C05467=1046.708,-58.246,426.994,169.791,33.093,156.253
C05468=1046.701,-58.495,427.006,169.789,33.092,156.253
C05469=1046.696,-58.746,427.017,169.787,33.091,156.252
C05470=1046.689,-58.995,427.029,169.784,33.090,156.252
C05471=1046.683,-59.245,427.041,169.782,33.089,156.252
C05472=1046.677,-59.495,427.054,169.780,33.088,156.252
C05473=1046.671,-59.744,427.065,169.778,33.088,156.252
C05474=1046.664,-59.993,427.077,169.776,33.086,156.252
C05475=1046.658,-60.243,427.090,169.774,33.085,156.252
C05476=1046.651,-60.493,427.102,169.772,33.085,156.252
C05477=1046.645,-60.742,427.114,169.769,33.084,156.252
C05478=1046.639,-60.992,427.126,169.767,33.082,156.252
C05479=1046.633,-61.242,427.137,169.765,33.081,156.252
C05480=1046.626,-61.491,427.149,169.763,33.081,156.251
C05481=1046.621,-61.741,427.162,169.761,33.080,156.251
C05482=1046.614,-61.991,427.174,169.759,33.079,156.251
C05483=1046.607,-62.240,427.186,169.757,33.078,156.251
C05484=1046.602,-62.489,427.198,169.755,33.077,156.251
C05485=1046.596,-62.740,427.209,169.752,33.076,156.251
C05486=1046.589,-62.989,427.221,169.750,33.075,156.251
C05487=1046.583,-63.239,427.234,169.748,33.074,156.251
C05488=1046.576,-63.489,427.246,169.746,33.073,156.251
C05489=1046.570,-63.737,427.257,169.744,33.072,156.251
C05490=1046.565,-63.988,427.269,169.742,33.071,156.251
C05491=1046.558,-64.238,427.281,169.739,33.070,156.250
C05492=1046.551,-64.487,427.293,169.738,33.069,156.250
C05493=1046.545,-64.736,427.305,169.736,33.068,156.250
C05494=1046.540,-64.986,427.316,169.734,33.067,156.250
C05495=1046.533,-65.236,427.328,169.732,33.066,156.250
C05496=1046.527,-65.485,427.340,169.730,33.065,156.250
C05497=1046.521,-65.735,427.353,169.728,33.065,156.250
C05498=1046.515,-65.985,427.364,169.725,33.064,156.250
C05499=1046.508,-66.235,427.376,169.723,33.062,156.250
C05500=1046.503,-66.484,427.388,169.721,33.061,156.250
C05501=1046.497,-66.734,427.399,169.719,33.061,156.250
C05502=1046.489,-67.016,427.413,169.716,33.060,156.250
C05503=1046.483,-67.299,427.426,169.714,33.058,156.249
C05504=1046.476,-67.581,427.440,169.712,33.057,156.249
C05505=1046.469,-67.863,427.453,169.709,33.057,156.249
C05506=1046.462,-68.113,427.465,169.707,33.056,156.249
C05507=1046.456,-68.362,427.476,169.705,33.055,156.249
C05508=1046.450,-68.612,427.487,169.703,33.054,156.249
C05509=1046.444,-68.862,427.500,169.701,33.053,156.249
C05510=1046.438,-69.111,427.511,169.698,33.052,156.249
C05511=1046.432,-69.361,427.523,169.696,33.051,156.249
C05512=1046.425,-69.611,427.535,169.694,33.050,156.249
C05513=1046.420,-69.860,427.546,169.692,33.049,156.249
C05514=1046.413,-70.110,427.558,169.690,33.049,156.248
C05515=1046.407,-70.360,427.569,169.688,33.048,156.248
C05516=1046.401,-70.609,427.581,169.685,33.047,156.248
C05517=1046.395,-70.859,427.593,169.683,33.046,156.248
C05518=1046.389,-71.108,427.604,169.681,33.045,156.248
C05519=1046.383,-71.358,427.616,169.679,33.044,156.248
C05520=1046.376,-71.608,427.628,169.677,33.043,156.248
C05521=1046.371,-71.857,427.640,169.674,33.042,156.248
C05522=1046.365,-72.107,427.651,169.672,33.041,156.248
C05523=1046.359,-72.356,427.663,169.670,33.040,156.248
C05524=1046.352,-72.607,427.674,169.669,33.040,156.248
C05525=1046.347,-72.856,427.686,169.667,33.039,156.248
C05526=1046.341,-73.106,427.697,169.665,33.038,156.248
C05527=1046.334,-73.356,427.709,169.662,33.037,156.248
C05528=1046.328,-73.605,427.720,169.660,33.036,156.247
C05529=1046.322,-73.855,427.731,169.658,33.035,156.247
C05530=1046.317,-74.104,427.744,169.656,33.035,156.247
C05531=1046.310,-74.355,427.755,169.654,33.034,156.247
C05532=1046.304,-74.603,427.766,169.651,33.033,156.247
C05533=1046.298,-74.854,427.778,169.649,33.032,156.247
C05534=1046.292,-75.104,427.789,169.647,33.031,156.247
C05535=1046.285,-75.352,427.800,169.645,33.030,156.247
C05536=1046.278,-75.603,427.811,169.643,33.030,156.247
C05537=1046.273,-75.852,427.822,169.640,33.029,156.247
C05538=1046.266,-76.102,427.834,169.638,33.028,156.247
C05539=1046.260,-76.351,427.845,169.636,33.028,156.247
C05540=1046.254,-76.601,427.856,169.634,33.027,156.247
C05541=1046.248,-76.850,427.868,169.632,33.026,156.247
C05542=1046.242,-77.100,427.879,169.629,33.025,156.247
C05543=1046.235,-77.351,427.890,169.627,33.024,156.247
C05544=1046.229,-77.599,427.902,169.625,33.024,156.247
C05545=1046.223,-77.850,427.913,169.623,33.023,156.247
C05546=1046.217,-78.099,427.924,169.620,33.022,156.247
C05547=1046.210,-78.349,427.936,169.618,33.021,156.246
C05548=1046.205,-78.598,427.947,169.616,33.021,156.246
C05549=1046.198,-78.848,427.958,169.614,33.020,156.246
C05550=1046.193,-79.098,427.969,169.612,33.020,156.246
C05551=1046.186,-79.348,427.980,169.609,33.019,156.246
C05552=1046.180,-79.597,427.992,169.607,33.018,156.246
C05553=1046.174,-79.847,428.003,169.605,33.017,156.246
C05554=1046.167,-80.096,428.013,169.603,33.016,156.246
C05555=1046.161,-80.346,428.025,169.601,33.016,156.246
C05556=1046.155,-80.596,428.035,169.599,33.015,156.246
C05557=1046.149,-80.846,428.047,169.597,33.014,156.246
C05558=1046.142,-81.095,428.058,169.595,33.014,156.246
C05559=1046.136,-81.345,428.069,169.592,33.013,156.246
C05560=1046.130,-81.594,428.080,169.590,33.012,156.246
C05561=1046.124,-81.845,428.091,169.588,33.012,156.246
C05562=1046.117,-82.094,428.101,169.586,33.011,156.246
C05563=1046.111,-82.344,428.113,169.583,33.011,156.246
C05564=1046.105,-82.593,428.123,169.581,33.010,156.246
C05565=1046.098,-82.843,428.134,169.579,33.009,156.246
C05566=1046.091,-83.127,428.147,169.576,33.009,156.246
C05567=1046.084,-83.412,428.160,169.574,33.008,156.246
C05568=1046.077,-83.697,428.172,169.571,33.007,156.246
C05569=1046.070,-83.981,428.184,169.569,33.007,156.246
C05570=1046.063,-84.231,428.196,169.566,33.006,156.246
C05571=1046.058,-84.480,428.206,169.564,33.006,156.246
C05572=1046.051,-84.730,428.217,169.562,33.005,156.246
C05573=1046.045,-84.980,428.228,169.560,33.005,156.246
C05574=1046.039,-85.229,428.239,169.557,33.004,156.246
C05575=1046.032,-85.479,428.249,169.555,33.003,156.246
C05576=1046.026,-85.729,428.260,169.553,33.003,156.246
C05577=1046.020,-85.979,428.272,169.551,33.002,156.246
C05578=1046.013,-86.228,428.282,169.548,33.002,156.246
C05579=1046.008,-86.477,428.293,169.546,33.001,156.246
C05580=1046.001,-86.728,428.304,169.544,33.000,156.246
C05581=1045.995,-86.977,428.314,169.542,33.000,156.246
C05582=1045.989,-87.227,428.326,169.540,32.999,156.246
C05583=1045.983,-87.477,428.336,169.538,32.999,156.245
C05584=1045.977,-87.726,428.346,169.536,32.998,156.246
C05585=1045.970,-87.977,428.357,169.533,32.997,156.245
C05586=1045.965,-88.226,428.368,169.531,32.997,156.246
C05587=1045.958,-88.475,428.378,169.529,32.996,156.245
C05588=1045.952,-88.725,428.390,169.527,32.996,156.246
C05589=1045.946,-88.975,428.400,169.524,32.995,156.245
C05590=1045.940,-89.224,428.411,169.522,32.995,156.245
C05591=1045.933,-89.474,428.422,169.520,32.994,156.245
C05592=1045.927,-89.724,428.433,169.518,32.994,156.245
C05593=1045.921,-89.974,428.442,169.515,32.993,156.245
C05594=1045.915,-90.224,428.454,169.513,32.993,156.245
C05595=1045.909,-90.473,428.465,169.511,32.992,156.245
C05596=1045.903,-90.722,428.475,169.508,32.992,156.245
C05597=1045.896,-90.973,428.486,169.506,32.991,156.245
C05598=1045.890,-91.222,428.496,169.504,32.991,156.245
C05599=1045.884,-91.472,428.507,169.502,32.990,156.245
C05600=1045.878,-91.722,428.518,169.499,32.990,156.245
C05601=1045.872,-91.971,428.528,169.497,32.989,156.245
C05602=1045.866,-92.221,428.539,169.495,32.989,156.245
C05603=1045.860,-92.470,428.550,169.493,32.988,156.245
C05604=1045.853,-92.721,428.560,169.490,32.988,156.245
C05605=1045.848,-92.970,428.571,169.488,32.987,156.245
C05606=1045.841,-93.219,428.581,169.486,32.987,156.245
C05607=1045.835,-93.469,428.592,169.483,32.986,156.245
C05608=1045.829,-93.720,428.602,169.481,32.986,156.245
C05609=1045.823,-93.969,428.613,169.479,32.985,156.245
C05610=1045.817,-94.218,428.623,169.477,32.985,156.245
C05611=1045.811,-94.468,428.633,169.475,32.984,156.245
C05612=1045.805,-94.718,428.644,169.473,32.983,156.245
C05613=1045.799,-94.968,428.655,169.471,32.983,156.245
C05614=1045.792,-95.217,428.665,169.468,32.982,156.245
C05615=1045.787,-95.467,428.676,169.466,32.982,156.245
C05616=1045.781,-95.716,428.686,169.464,32.982,156.245
C05617=1045.775,-95.966,428.697,169.462,32.981,156.245
C05618=1045.769,-96.217,428.707,169.459,32.981,156.245
C05619=1045.762,-96.466,428.718,169.457,32.980,156.245
C05620=1045.757,-96.716,428.728,169.455,32.980,156.245
C05621=1045.750,-96.965,428.738,169.452,32.980,156.245
C05622=1045.745,-97.215,428.749,169.450,32.979,156.245
C05623=1045.738,-97.465,428.759,169.448,32.979,156.245
C05624=1045.732,-97.715,428.770,169.446,32.978,156.245
C05625=1045.726,-97.964,428.779,169.443,32.977,156.245
C05626=1045.720,-98.214,428.790,169.441,32.977,156.245
C05627=1045.714,-98.463,428.800,169.439,32.977,156.246
C05628=1045.707,-98.714,428.810,169.436,32.977,156.246
C05629=1045.701,-98.963,428.821,169.434,32.977,156.246
C05630=1045.695,-99.250,428.832,169.431,32.976,156.246
C05631=1045.687,-99.536,428.844,169.429,32.975,156.246
C05632=1045.680,-99.824,428.855,169.426,32.975,156.246
C05633=1045.673,-100.111,428.868,169.423,32.975,156.246
C05634=1045.667,-100.360,428.877,169.421,32.974,156.246
C05635=1045.660,-100.610,428.888,169.419,32.974,156.246
C05636=1045.655,-100.860,428.898,169.416,32.974,156.246
C05637=1045.648,-101.109,428.908,169.415,32.973,156.246
C05638=1045.642,-101.359,428.918,169.413,32.973,156.246
C05639=1045.636,-101.608,428.929,169.410,32.973,156.246
C05640=1045.629,-101.859,428.939,169.408,32.972,156.246
C05641=1045.623,-102.108,428.949,169.406,32.972,156.246
C05642=1045.618,-102.358,428.959,169.403,32.972,156.246
C05643=1045.611,-102.608,428.969,169.401,32.971,156.246
C05644=1045.605,-102.857,428.979,169.399,32.971,156.246
C05645=1045.600,-103.107,428.989,169.397,32.971,156.246
C05646=1045.593,-103.356,428.999,169.394,32.971,156.246
C05647=1045.587,-103.606,429.009,169.392,32.970,156.246
C05648=1045.581,-103.856,429.018,169.390,32.970,156.246
C05649=1045.575,-104.105,429.029,169.387,32.969,156.246
C05650=1045.569,-104.355,429.039,169.385,32.969,156.246
C05651=1045.562,-104.606,429.049,169.383,32.969,156.246
C05652=1045.556,-104.855,429.060,169.380,32.969,156.246
C05653=1045.550,-105.105,429.069,169.378,32.969,156.246
C05654=1045.544,-105.355,429.079,169.376,32.968,156.246
C05655=1045.537,-105.604,429.089,169.373,32.968,156.246
C05656=1045.532,-105.854,429.099,169.371,32.968,156.247
C05657=1045.526,-106.104,429.109,169.369,32.968,156.247
C05658=1045.520,-106.354,429.118,169.366,32.967,156.247
C05659=1045.513,-106.603,429.129,169.364,32.967,156.247
C05660=1045.507,-106.853,429.138,169.362,32.966,156.247
C05661=1045.502,-107.103,429.148,169.359,32.966,156.247
C05662=1045.495,-107.352,429.158,169.357,32.966,156.247
C05663=1045.489,-107.602,429.168,169.355,32.966,156.247
C05664=1045.483,-107.851,429.178,169.353,32.966,156.247
C05665=1045.477,-108.101,429.187,169.351,32.965,156.247
C05666=1045.470,-108.351,429.197,169.349,32.966,156.247
C05667=1045.465,-108.601,429.208,169.346,32.965,156.247
C05668=1045.459,-108.850,429.217,169.344,32.965,156.247
C05669=1045.452,-109.100,429.227,169.341,32.965,156.247
C05670=1045.446,-109.350,429.237,169.339,32.965,156.247
C05671=1045.440,-109.600,429.246,169.337,32.965,156.247
C05672=1045.434,-109.850,429.256,169.334,32.964,156.247
C05673=1045.427,-110.099,429.266,169.332,32.964,156.247
C05674=1045.421,-110.348,429.275,169.330,32.964,156.247
C05675=1045.415,-110.598,429.285,169.327,32.964,156.247
C05676=1045.409,-110.848,429.295,169.325,32.963,156.248
C05677=1045.403,-111.098,429.305,169.323,32.964,156.248
C05678=1045.397,-111.348,429.314,169.320,32.964,156.248
C05679=1045.391,-111.598,429.324,169.318,32.963,156.248
C05680=1045.385,-111.848,429.333,169.316,32.963,156.248
C05681=1045.379,-112.097,429.343,169.313,32.963,156.248
C05682=1045.373,-112.347,429.353,169.311,32.963,156.248
C05683=1045.366,-112.597,429.362,169.308,32.962,156.248
C05684=1045.360,-112.846,429.372,169.306,32.962,156.248
C05685=1045.354,-113.096,429.382,169.304,32.963,156.248
C05686=1045.348,-113.346,429.392,169.301,32.962,156.248
C05687=1045.342,-113.595,429.401,169.299,32.962,156.248
C05688=1045.336,-113.845,429.410,169.297,32.962,156.248
C05689=1045.330,-114.094,429.420,169.295,32.962,156.248
C05690=1045.323,-114.344,429.430,169.293,32.962,156.248
C05691=1045.317,-114.594,429.439,169.291,32.962,156.249
C05692=1045.311,-114.844,429.449,169.288,32.962,156.249
C05693=1045.305,-115.094,429.458,169.286,32.962,156.249
C05694=1045.298,-115.380,429.469,169.283,32.961,156.249
C05695=1045.291,-115.665,429.480,169.280,32.962,156.249
C05696=1045.284,-115.952,429.491,169.278,32.961,156.249
C05697=1045.277,-116.237,429.501,169.275,32.961,156.249
C05698=1045.271,-116.487,429.511,169.273,32.962,156.249
C05699=1045.265,-116.736,429.520,169.270,32.961,156.249
C05700=1045.259,-116.986,429.530,169.268,32.961,156.249
C05701=1045.253,-117.237,429.539,169.266,32.962,156.249
C05702=1045.247,-117.486,429.548,169.263,32.961,156.250
C05703=1045.240,-117.736,429.558,169.261,32.961,156.250
C05704=1045.235,-117.985,429.567,169.258,32.961,156.250
C05705=1045.229,-118.235,429.577,169.256,32.961,156.250
C05706=1045.223,-118.485,429.586,169.254,32.961,156.250
C05707=1045.216,-118.734,429.595,169.251,32.961,156.250
C05708=1045.210,-118.985,429.604,169.249,32.961,156.250
C05709=1045.204,-119.235,429.614,169.247,32.961,156.250
C05710=1045.198,-119.484,429.623,169.244,32.961,156.250
C05711=1045.192,-119.733,429.632,169.242,32.961,156.250
C05712=1045.186,-119.983,429.642,169.239,32.961,156.250
C05713=1045.180,-120.234,429.651,169.237,32.961,156.251
C05714=1045.174,-120.483,429.660,169.235,32.961,156.251
C05715=1045.167,-120.732,429.669,169.233,32.961,156.251
C05716=1045.161,-120.982,429.679,169.231,32.961,156.251
C05717=1045.155,-121.232,429.688,169.228,32.961,156.251
C05718=1045.149,-121.482,429.697,169.226,32.962,156.251
C05719=1045.143,-121.732,429.707,169.224,32.961,156.251
C05720=1045.137,-121.981,429.716,169.221,32.962,156.251
C05721=1045.130,-122.231,429.725,169.219,32.961,156.251
C05722=1045.125,-122.481,429.734,169.217,32.961,156.251
C05723=1045.118,-122.731,429.743,169.214,32.962,156.251
C05724=1045.113,-122.980,429.752,169.212,32.961,156.252
C05725=1045.107,-123.230,429.761,169.209,32.962,156.252
C05726=1045.101,-123.480,429.771,169.207,32.962,156.252
C05727=1045.094,-123.730,429.780,169.205,32.962,156.252
C05728=1045.089,-123.979,429.788,169.202,32.962,156.252
C05729=1045.083,-124.229,429.798,169.200,32.962,156.252
C05730=1045.076,-124.479,429.807,169.197,32.962,156.252
C05731=1045.070,-124.729,429.816,169.195,32.962,156.252
C05732=1045.064,-124.978,429.825,169.193,32.962,156.252
C05733=1045.058,-125.228,429.834,169.190,32.963,156.253
C05734=1045.052,-125.478,429.843,169.188,32.962,156.253
C05735=1045.045,-125.728,429.852,169.185,32.963,156.253
C05736=1045.040,-125.978,429.861,169.183,32.963,156.253
C05737=1045.034,-126.227,429.870,169.181,32.963,156.253
C05738=1045.027,-126.478,429.878,169.178,32.963,156.253
C05739=1045.022,-126.727,429.888,169.176,32.963,156.253
C05740=1045.015,-126.976,429.897,169.174,32.964,156.253
C05741=1045.009,-127.227,429.906,169.172,32.964,156.254
C05742=1045.003,-127.476,429.915,169.170,32.964,156.254
C05743=1044.997,-127.726,429.924,169.167,32.964,156.254
C05744=1044.992,-127.975,429.933,169.165,32.964,156.254
C05745=1044.986,-128.225,429.943,169.163,32.963,156.254
C05746=1044.982,-128.475,429.953,169.161,32.962,156.254
C05747=1044.980,-128.725,429.965,169.159,32.961,156.253
C05748=1044.978,-128.975,429.976,169.157,32.959,156.253
C05749=1044.977,-129.225,429.989,169.155,32.957,156.253
C05750=1044.977,-129.475,430.001,169.153,32.954,156.252
C05751=1044.978,-129.725,430.015,169.152,32.951,156.252
C05752=1044.979,-129.976,430.029,169.150,32.947,156.251
C05753=1044.982,-130.225,430.043,169.149,32.943,156.251
C05754=1044.986,-130.476,430.059,169.148,32.938,156.250
C05755=1044.990,-130.727,430.075,169.147,32.933,156.249
C05756=1044.995,-130.977,430.092,169.146,32.927,156.248
C05757=1045.002,-131.227,430.109,169.145,32.921,156.247
C05758=1044.646,-131.251,429.866,169.099,33.102,156.280
C05759=1044.641,-131.000,429.849,169.100,33.108,156.281
C05760=1044.635,-130.751,429.832,169.101,33.114,156.282
C05761=1044.631,-130.500,429.816,169.102,33.119,156.283
C05762=1044.627,-130.249,429.801,169.103,33.124,156.283
C05763=1044.624,-129.999,429.786,169.104,33.128,156.284
C05764=1044.622,-129.749,429.771,169.105,33.131,156.285
C05765=1044.622,-129.499,429.758,169.107,33.135,156.285
C05766=1044.622,-129.248,429.745,169.108,33.138,156.285
C05767=1044.623,-128.998,429.732,169.110,33.140,156.286
C05768=1044.625,-128.749,429.721,169.112,33.142,156.286
C05769=1044.627,-128.498,429.709,169.114,33.144,156.286
C05770=1044.631,-128.249,429.699,169.116,33.145,156.286
C05771=1044.636,-127.999,429.689,169.118,33.145,156.286
C05772=1044.641,-127.749,429.680,169.121,33.145,156.286
C05773=1044.648,-127.500,429.671,169.123,33.145,156.286
C05774=1044.653,-127.251,429.662,169.125,33.145,156.286
C05775=1044.659,-127.000,429.653,169.128,33.144,156.286
C05776=1044.666,-126.751,429.644,169.130,33.145,156.286
C05777=1044.671,-126.501,429.636,169.133,33.144,156.286
C05778=1044.677,-126.251,429.626,169.135,33.144,156.286
C05779=1044.684,-126.001,429.618,169.138,33.144,156.285
C05780=1044.690,-125.751,429.608,169.140,33.144,156.285
C05781=1044.696,-125.502,429.600,169.142,33.144,156.285
C05782=1044.702,-125.252,429.591,169.145,33.143,156.285
C05783=1044.709,-125.002,429.581,169.147,33.143,156.285
C05784=1044.714,-124.753,429.573,169.149,33.143,156.285
C05785=1044.721,-124.503,429.564,169.151,33.143,156.285
C05786=1044.727,-124.253,429.554,169.153,33.143,156.285
C05787=1044.733,-124.003,429.545,169.156,33.143,156.285
C05788=1044.738,-123.754,429.536,169.158,33.143,156.285
C05789=1044.745,-123.504,429.527,169.161,33.142,156.284
C05790=1044.751,-123.254,429.518,169.163,33.143,156.284
C05791=1044.757,-123.004,429.509,169.165,33.142,156.284
C05792=1044.763,-122.755,429.500,169.168,33.142,156.284
C05793=1044.769,-122.505,429.491,169.170,33.142,156.284
C05794=1044.775,-122.255,429.481,169.173,33.142,156.284
C05795=1044.782,-122.005,429.472,169.175,33.142,156.284
C05796=1044.787,-121.756,429.464,169.177,33.142,156.284
C05797=1044.793,-121.506,429.454,169.180,33.142,156.284
C05798=1044.799,-121.256,429.445,169.182,33.142,156.283
C05799=1044.806,-121.006,429.435,169.185,33.142,156.283
C05800=1044.812,-120.756,429.426,169.187,33.142,156.283
C05801=1044.817,-120.507,429.417,169.189,33.142,156.283
C05802=1044.824,-120.257,429.408,169.192,33.141,156.283
C05803=1044.830,-120.008,429.398,169.194,33.142,156.283
C05804=1044.836,-119.758,429.389,169.197,33.141,156.283
C05805=1044.842,-119.507,429.380,169.199,33.141,156.283
C05806=1044.848,-119.258,429.371,169.201,33.142,156.283
C05807=1044.854,-119.008,429.361,169.204,33.141,156.283
C05808=1044.860,-118.759,429.352,169.206,33.141,156.283
C05809=1044.866,-118.509,429.342,169.208,33.142,156.282
C05810=1044.873,-118.259,429.333,169.210,33.141,156.282
C05811=1044.879,-118.009,429.324,169.212,33.141,156.282
C05812=1044.885,-117.760,429.315,169.215,33.141,156.282
C05813=1044.891,-117.510,429.306,169.217,33.141,156.282
C05814=1044.897,-117.260,429.296,169.220,33.141,156.282
C05815=1044.903,-117.010,429.286,169.222,33.141,156.282
C05816=1044.909,-116.761,429.277,169.224,33.141,156.282
C05817=1044.915,-116.511,429.267,169.227,33.141,156.282
C05818=1044.922,-116.261,429.258,169.229,33.141,156.282
C05819=1044.929,-115.975,429.248,169.232,33.141,156.282
C05820=1044.936,-115.689,429.236,169.235,33.141,156.281
C05821=1044.943,-115.403,429.226,169.237,33.141,156.281
C05822=1044.949,-115.118,429.215,169.240,33.141,156.281
C05823=1044.956,-114.868,429.205,169.242,33.141,156.281
C05824=1044.962,-114.618,429.196,169.245,33.142,156.281
C05825=1044.968,-114.369,429.186,169.247,33.141,156.281
C05826=1044.974,-114.119,429.176,169.249,33.141,156.281
C05827=1044.980,-113.869,429.167,169.252,33.142,156.281
C05828=1044.986,-113.619,429.157,169.254,33.142,156.281
C05829=1044.992,-113.370,429.148,169.257,33.142,156.281
C05830=1044.998,-113.120,429.139,169.259,33.142,156.281
C05831=1045.004,-112.870,429.129,169.261,33.142,156.281
C05832=1045.011,-112.621,429.119,169.264,33.142,156.281
C05833=1045.017,-112.371,429.110,169.266,33.142,156.281
C05834=1045.023,-112.121,429.100,169.268,33.143,156.280
C05835=1045.029,-111.871,429.091,169.270,33.142,156.280
C05836=1045.035,-111.621,429.081,169.272,33.142,156.280
C05837=1045.041,-111.371,429.071,169.275,33.143,156.280
C05838=1045.047,-111.122,429.061,169.277,33.143,156.280
C05839=1045.053,-110.872,429.052,169.279,33.143,156.280
C05840=1045.059,-110.622,429.042,169.282,33.143,156.280
C05841=1045.066,-110.373,429.032,169.284,33.143,156.280
C05842=1045.072,-110.123,429.022,169.286,33.143,156.280
C05843=1045.078,-109.873,429.013,169.289,33.143,156.280
C05844=1045.084,-109.623,429.003,169.291,33.143,156.280
C05845=1045.090,-109.374,428.994,169.293,33.144,156.280
C05846=1045.096,-109.124,428.984,169.296,33.144,156.280
C05847=1045.103,-108.874,428.975,169.298,33.144,156.280
C05848=1045.108,-108.624,428.964,169.301,33.144,156.280
C05849=1045.115,-108.375,428.954,169.303,33.145,156.280
C05850=1045.121,-108.125,428.945,169.305,33.145,156.280
C05851=1045.127,-107.875,428.935,169.308,33.144,156.279
C05852=1045.133,-107.625,428.925,169.310,33.144,156.279
C05853=1045.140,-107.376,428.915,169.312,33.145,156.279
C05854=1045.146,-107.126,428.906,169.315,33.145,156.279
C05855=1045.151,-106.876,428.895,169.317,33.145,156.279
C05856=1045.157,-106.626,428.886,169.319,33.145,156.279
C05857=1045.164,-106.377,428.876,169.322,33.146,156.279
C05858=1045.170,-106.127,428.866,169.324,33.146,156.279
C05859=1045.175,-105.877,428.856,169.326,33.146,156.279
C05860=1045.182,-105.628,428.846,169.329,33.146,156.279
C05861=1045.188,-105.378,428.836,169.331,33.146,156.279
C05862=1045.194,-105.129,428.826,169.333,33.147,156.279
C05863=1045.200,-104.878,428.816,169.335,33.147,156.279
C05864=1045.206,-104.629,428.806,169.337,33.148,156.279
C05865=1045.212,-104.379,428.796,169.339,33.148,156.279
C05866=1045.219,-104.129,428.787,169.342,33.148,156.279
C05867=1045.225,-103.879,428.776,169.344,33.148,156.279
C05868=1045.231,-103.630,428.766,169.346,33.148,156.279
C05869=1045.237,-103.380,428.756,169.349,33.149,156.279
C05870=1045.243,-103.130,428.746,169.351,33.149,156.279
C05871=1045.249,-102.881,428.736,169.353,33.149,156.279
C05872=1045.256,-102.631,428.726,169.356,33.149,156.278
C05873=1045.262,-102.382,428.716,169.358,33.150,156.278
C05874=1045.267,-102.132,428.705,169.360,33.150,156.278
C05875=1045.274,-101.882,428.696,169.363,33.151,156.278
C05876=1045.280,-101.632,428.686,169.365,33.151,156.278
C05877=1045.286,-101.382,428.675,169.367,33.151,156.278
C05878=1045.292,-101.133,428.665,169.370,33.151,156.278
C05879=1045.299,-100.883,428.655,169.372,33.151,156.278
C05880=1045.304,-100.633,428.645,169.374,33.152,156.278
C05881=1045.311,-100.384,428.635,169.377,33.152,156.278
C05882=1045.317,-100.134,428.625,169.379,33.153,156.278
C05883=1045.324,-99.847,428.613,169.382,33.153,156.278
C05884=1045.331,-99.560,428.601,169.384,33.153,156.278
C05885=1045.339,-99.273,428.589,169.387,33.153,156.278
C05886=1045.345,-98.986,428.578,169.390,33.154,156.278
C05887=1045.351,-98.737,428.568,169.392,33.155,156.278
C05888=1045.358,-98.487,428.558,169.394,33.155,156.278
C05889=1045.364,-98.237,428.547,169.397,33.155,156.278
C05890=1045.370,-97.987,428.537,169.399,33.155,156.278
C05891=1045.376,-97.738,428.527,169.400,33.155,156.278
C05892=1045.382,-97.489,428.516,169.403,33.156,156.278
C05893=1045.389,-97.238,428.506,169.405,33.156,156.278
C05894=1045.395,-96.989,428.495,169.407,33.157,156.278
C05895=1045.401,-96.739,428.486,169.410,33.158,156.278
C05896=1045.406,-96.489,428.475,169.412,33.158,156.278
C05897=1045.412,-96.240,428.464,169.414,33.158,156.278
C05898=1045.418,-95.990,428.454,169.417,33.159,156.278
C05899=1045.425,-95.740,428.443,169.419,33.159,156.278
C05900=1045.431,-95.491,428.433,169.421,33.159,156.278
C05901=1045.437,-95.241,428.423,169.423,33.160,156.278
C05902=1045.443,-94.991,428.412,169.426,33.160,156.278
C05903=1045.449,-94.742,428.402,169.428,33.161,156.278
C05904=1045.455,-94.491,428.391,169.430,33.161,156.278
C05905=1045.461,-94.242,428.381,169.433,33.161,156.278
C05906=1045.467,-93.992,428.370,169.435,33.162,156.278
C05907=1045.474,-93.743,428.360,169.437,33.162,156.278
C05908=1045.480,-93.493,428.349,169.439,33.163,156.278
C05909=1045.485,-93.243,428.338,169.442,33.164,156.278
C05910=1045.492,-92.994,428.328,169.444,33.164,156.278
C05911=1045.498,-92.744,428.317,169.446,33.165,156.278
C05912=1045.504,-92.494,428.307,169.449,33.165,156.278
C05913=1045.510,-92.244,428.296,169.451,33.166,156.278
C05914=1045.516,-91.995,428.285,169.453,33.166,156.278
C05915=1045.522,-91.746,428.275,169.456,33.167,156.278
C05916=1045.528,-91.495,428.264,169.458,33.167,156.278
C05917=1045.534,-91.245,428.254,169.460,33.167,156.278
C05918=1045.541,-90.996,428.243,169.462,33.168,156.278
C05919=1045.547,-90.746,428.232,169.465,33.168,156.278
C05920=1045.553,-90.497,428.222,169.467,33.169,156.278
C05921=1045.559,-90.247,428.211,169.468,33.169,156.278
C05922=1045.565,-89.997,428.201,169.470,33.170,156.278
C05923=1045.572,-89.747,428.190,169.473,33.170,156.278
C05924=1045.577,-89.498,428.179,169.475,33.171,156.278
C05925=1045.583,-89.248,428.168,169.477,33.171,156.278
C05926=1045.590,-88.999,428.158,169.480,33.172,156.278
C05927=1045.596,-88.749,428.147,169.482,33.172,156.278
C05928=1045.602,-88.500,428.136,169.484,33.173,156.278
C05929=1045.609,-88.250,428.125,169.486,33.173,156.278
C05930=1045.614,-88.000,428.115,169.489,33.174,156.278
C05931=1045.621,-87.749,428.104,169.491,33.174,156.278
C05932=1045.627,-87.500,428.094,169.493,33.175,156.278
C05933=1045.633,-87.251,428.083,169.496,33.175,156.278
C05934=1045.639,-87.000,428.072,169.498,33.176,156.278
C05935=1045.646,-86.751,428.061,169.500,33.176,156.278
C05936=1045.651,-86.502,428.050,169.502,33.177,156.278
C05937=1045.658,-86.252,428.039,169.505,33.178,156.278
C05938=1045.664,-86.002,428.029,169.507,33.178,156.278
C05939=1045.670,-85.752,428.018,169.509,33.179,156.278
C05940=1045.676,-85.503,428.007,169.511,33.179,156.278
C05941=1045.683,-85.254,427.996,169.514,33.180,156.278
C05942=1045.689,-85.003,427.985,169.516,33.180,156.278
C05943=1045.695,-84.754,427.974,169.518,33.181,156.278
C05944=1045.702,-84.504,427.964,169.521,33.182,156.278
C05945=1045.708,-84.255,427.953,169.523,33.182,156.278
C05946=1045.714,-84.004,427.942,169.525,33.183,156.278
C05947=1045.721,-83.720,427.929,169.528,33.183,156.278
C05948=1045.728,-83.436,427.917,169.530,33.184,156.278
C05949=1045.735,-83.151,427.904,169.533,33.185,156.278
C05950=1045.742,-82.866,427.892,169.535,33.185,156.278
C05951=1045.749,-82.616,427.881,169.538,33.186,156.278
C05952=1045.755,-82.367,427.870,169.539,33.186,156.278
C05953=1045.761,-82.117,427.859,169.541,33.187,156.278
C05954=1045.768,-81.868,427.848,169.543,33.187,156.278
C05955=1045.774,-81.618,427.837,169.546,33.188,156.278
C05956=1045.780,-81.369,427.826,169.548,33.188,156.278
C05957=1045.786,-81.118,427.815,169.550,33.189,156.278
C05958=1045.793,-80.869,427.805,169.552,33.190,156.278
C05959=1045.799,-80.619,427.793,169.555,33.190,156.278
C05960=1045.805,-80.369,427.782,169.557,33.191,156.278
C05961=1045.812,-80.120,427.770,169.559,33.192,156.279
C05962=1045.818,-79.871,427.760,169.561,33.192,156.278
C05963=1045.824,-79.621,427.749,169.564,33.193,156.279
C05964=1045.830,-79.371,427.738,169.566,33.194,156.279
C05965=1045.836,-79.121,427.727,169.568,33.194,156.279
C05966=1045.843,-78.872,427.715,169.570,33.195,156.279
C05967=1045.849,-78.622,427.704,169.573,33.196,156.279
C05968=1045.855,-78.372,427.693,169.575,33.197,156.279
C05969=1045.861,-78.122,427.682,169.577,33.197,156.279
C05970=1045.867,-77.873,427.670,169.579,33.198,156.279
C05971=1045.873,-77.623,427.659,169.582,33.198,156.279
C05972=1045.879,-77.374,427.648,169.584,33.199,156.279
C05973=1045.886,-77.124,427.636,169.586,33.200,156.279
C05974=1045.891,-76.874,427.625,169.588,33.201,156.279
C05975=1045.898,-76.624,427.614,169.590,33.202,156.279
C05976=1045.904,-76.374,427.603,169.593,33.202,156.279
C05977=1045.910,-76.125,427.591,169.595,33.203,156.279
C05978=1045.917,-75.875,427.580,169.597,33.204,156.279
C05979=1045.923,-75.626,427.568,169.599,33.204,156.279
C05980=1045.930,-75.376,427.558,169.602,33.205,156.279
C05981=1045.935,-75.127,427.547,169.604,33.206,156.279
C05982=1045.942,-74.877,427.535,169.606,33.206,156.279
C05983=1045.948,-74.627,427.524,169.608,33.207,156.279
C05984=1045.954,-74.378,427.513,169.610,33.208,156.280
C05985=1045.961,-74.128,427.501,169.613,33.209,156.280
C05986=1045.966,-73.878,427.490,169.614,33.210,156.280
C05987=1045.972,-73.629,427.477,169.616,33.210,156.280
C05988=1045.978,-73.379,427.467,169.618,33.211,156.280
C05989=1045.985,-73.130,427.455,169.620,33.212,156.280
C05990=1045.991,-72.879,427.443,169.623,33.213,156.280
C05991=1045.996,-72.630,427.431,169.625,33.214,156.280
C05992=1046.003,-72.380,427.420,169.627,33.215,156.280
C05993=1046.009,-72.131,427.408,169.629,33.215,156.280
C05994=1046.015,-71.881,427.397,169.631,33.216,156.280
C05995=1046.020,-71.632,427.385,169.633,33.217,156.280
C05996=1046.027,-71.382,427.374,169.636,33.218,156.280
C05997=1046.033,-71.132,427.362,169.638,33.219,156.280
C05998=1046.039,-70.882,427.351,169.640,33.220,156.280
C05999=1046.045,-70.633,427.338,169.642,33.220,156.281
C06000=1046.051,-70.383,427.327,169.644,33.221,156.281
C06001=1046.057,-70.134,427.315,169.647,33.222,156.281
C06002=1046.064,-69.883,427.304,169.649,33.223,156.281
C06003=1046.069,-69.634,427.292,169.651,33.224,156.281
C06004=1046.076,-69.385,427.280,169.653,33.225,156.281
C06005=1046.082,-69.134,427.269,169.655,33.226,156.281
C06006=1046.088,-68.886,427.257,169.657,33.227,156.281
C06007=1046.094,-68.635,427.245,169.660,33.228,156.281
C06008=1046.100,-68.386,427.234,169.662,33.228,156.281
C06009=1046.106,-68.137,427.222,169.664,33.229,156.281
C06010=1046.113,-67.886,427.211,169.666,33.230,156.281
C06011=1046.120,-67.604,427.197,169.669,33.231,156.281
C06012=1046.127,-67.322,427.184,169.671,33.232,156.282
C06013=1046.134,-67.040,427.170,169.673,33.233,156.282
C06014=1046.140,-66.757,427.157,169.676,33.234,156.282
C06015=1046.147,-66.507,427.145,169.678,33.235,156.282
C06016=1046.152,-66.258,427.134,169.680,33.236,156.282
C06017=1046.159,-66.008,427.122,169.682,33.237,156.282
C06018=1046.165,-65.758,427.110,169.685,33.238,156.282
C06019=1046.171,-65.509,427.097,169.687,33.239,156.282
C06020=1046.177,-65.259,427.086,169.689,33.240,156.282
C06021=1046.184,-65.009,427.074,169.691,33.240,156.282
C06022=1046.190,-64.760,427.062,169.693,33.241,156.282
C06023=1046.196,-64.510,427.050,169.695,33.242,156.282
C06024=1046.202,-64.261,427.039,169.697,33.243,156.283
C06025=1046.209,-64.011,427.027,169.699,33.244,156.283
C06026=1046.214,-63.761,427.014,169.701,33.245,156.283
C06027=1046.221,-63.511,427.003,169.703,33.246,156.283
C06028=1046.227,-63.262,426.992,169.705,33.247,156.283
C06029=1046.233,-63.012,426.979,169.707,33.248,156.283
C06030=1046.239,-62.763,426.967,169.709,33.248,156.283
C06031=1046.246,-62.513,426.955,169.712,33.250,156.283
C06032=1046.251,-62.264,426.943,169.714,33.251,156.283
C06033=1046.258,-62.014,426.931,169.716,33.252,156.283
C06034=1046.264,-61.764,426.920,169.718,33.252,156.283
C06035=1046.270,-61.514,426.907,169.720,33.253,156.284
C06036=1046.277,-61.265,426.895,169.722,33.254,156.284
C06037=1046.283,-61.016,426.884,169.725,33.255,156.284
C06038=1046.289,-60.766,426.871,169.727,33.256,156.284
C06039=1046.296,-60.516,426.859,169.729,33.257,156.284
C06040=1046.302,-60.267,426.847,169.731,33.258,156.284
C06041=1046.308,-60.016,426.835,169.733,33.259,156.284
C06042=1046.314,-59.767,426.823,169.735,33.260,156.284
C06043=1046.320,-59.518,426.812,169.737,33.261,156.284
C06044=1046.326,-59.268,426.799,169.740,33.262,156.284
C06045=1046.333,-59.018,426.787,169.742,33.263,156.284
C06046=1046.340,-58.769,426.775,169.744,33.263,156.285
C06047=1046.346,-58.519,426.763,169.746,33.265,156.285
C06048=1046.352,-58.269,426.751,169.748,33.266,156.285
C06049=1046.359,-58.020,426.739,169.750,33.266,156.285
C06050=1046.365,-57.770,426.726,169.752,33.267,156.285
C06051=1046.371,-57.521,426.715,169.755,33.268,156.285
C06052=1046.377,-57.271,426.702,169.757,33.270,156.285
C06053=1046.383,-57.021,426.690,169.759,33.270,156.285
C06054=1046.390,-56.772,426.678,169.761,33.271,156.285
C06055=1046.396,-56.522,426.666,169.763,33.272,156.285
C06056=1046.403,-56.272,426.654,169.765,33.273,156.286
C06057=1046.409,-56.023,426.642,169.767,33.274,156.286
C06058=1046.415,-55.773,426.629,169.769,33.275,156.286
C06059=1046.422,-55.523,426.617,169.772,33.276,156.286
C06060=1046.428,-55.274,426.605,169.774,33.277,156.286
C06061=1046.434,-55.024,426.593,169.776,33.278,156.286
C06062=1046.441,-54.774,426.581,169.778,33.279,156.286
C06063=1046.447,-54.525,426.568,169.780,33.280,156.286
C06064=1046.453,-54.276,426.557,169.782,33.281,156.286
C06065=1046.459,-54.026,426.544,169.784,33.282,156.286
C06066=1046.465,-53.776,426.532,169.786,33.283,156.287
C06067=1046.472,-53.527,426.519,169.789,33.284,156.287
C06068=1046.478,-53.277,426.507,169.790,33.285,156.287
C06069=1046.485,-53.028,426.495,169.792,33.286,156.287
C06070=1046.491,-52.778,426.482,169.794,33.287,156.287
C06071=1046.498,-52.528,426.470,169.796,33.288,156.287
C06072=1046.504,-52.279,426.458,169.798,33.289,156.287
C06073=1046.510,-52.029,426.446,169.800,33.290,156.287
C06074=1046.517,-51.780,426.433,169.802,33.291,156.287
C06075=1046.524,-51.498,426.420,169.805,33.292,156.287
C06076=1046.531,-51.217,426.405,169.807,33.293,156.288
C06077=1046.539,-50.936,426.392,169.810,33.294,156.288
C06078=1046.546,-50.655,426.378,169.812,33.295,156.288
C06079=1046.552,-50.405,426.365,169.814,33.296,156.288
C06080=1046.558,-50.156,426.353,169.816,33.298,156.288
C06081=1046.564,-49.906,426.341,169.818,33.298,156.288
C06082=1046.570,-49.657,426.327,169.820,33.300,156.288
C06083=1046.576,-49.407,426.315,169.822,33.301,156.288
C06084=1046.583,-49.157,426.303,169.824,33.302,156.289
C06085=1046.589,-48.907,426.290,169.826,33.303,156.289
C06086=1046.595,-48.658,426.277,169.829,33.304,156.289
C06087=1046.601,-48.408,426.264,169.831,33.306,156.289
C06088=1046.608,-48.159,426.252,169.833,33.307,156.289
C06089=1046.614,-47.909,426.239,169.835,33.308,156.289
C06090=1046.620,-47.660,426.227,169.837,33.309,156.289
C06091=1046.626,-47.410,426.213,169.839,33.310,156.290
C06092=1046.633,-47.161,426.201,169.841,33.311,156.290
C06093=1046.639,-46.911,426.189,169.843,33.312,156.290
C06094=1046.645,-46.661,426.175,169.845,33.313,156.290
C06095=1046.651,-46.411,426.163,169.847,33.315,156.290
C06096=1046.658,-46.161,426.151,169.849,33.315,156.290
C06097=1046.664,-45.912,426.137,169.851,33.317,156.290
C06098=1046.670,-45.662,426.125,169.853,33.318,156.290
C06099=1046.676,-45.413,426.112,169.855,33.319,156.291
C06100=1046.682,-45.163,426.099,169.857,33.321,156.291
C06101=1046.689,-44.914,426.087,169.859,33.321,156.291
C06102=1046.695,-44.664,426.074,169.862,33.323,156.291
C06103=1046.701,-44.414,426.061,169.864,33.324,156.291
C06104=1046.707,-44.165,426.048,169.866,33.325,156.291
C06105=1046.713,-43.915,426.035,169.868,33.326,156.291
C06106=1046.720,-43.666,426.023,169.870,33.327,156.292
C06107=1046.726,-43.416,426.010,169.872,33.329,156.292
C06108=1046.733,-43.166,425.997,169.874,33.330,156.292
C06109=1046.739,-42.917,425.984,169.876,33.331,156.292
C06110=1046.745,-42.667,425.971,169.878,33.332,156.292
C06111=1046.751,-42.418,425.959,169.880,33.333,156.292
C06112=1046.758,-42.168,425.945,169.882,33.335,156.292
C06113=1046.764,-41.919,425.933,169.884,33.335,156.292
C06114=1046.770,-41.669,425.920,169.886,33.337,156.293
C06115=1046.776,-41.419,425.907,169.888,33.338,156.293
C06116=1046.783,-41.170,425.894,169.890,33.339,156.293
C06117=1046.789,-40.921,425.881,169.892,33.340,156.293
C06118=1046.795,-40.671,425.868,169.894,33.341,156.293
C06119=1046.802,-40.421,425.855,169.896,33.343,156.293
C06120=1046.807,-40.171,425.842,169.898,33.344,156.293
C06121=1046.814,-39.923,425.830,169.900,33.345,156.294
C06122=1046.821,-39.672,425.817,169.902,33.346,156.294
C06123=1046.827,-39.423,425.804,169.904,33.347,156.294
C06124=1046.833,-39.173,425.790,169.907,33.349,156.294
C06125=1046.839,-38.924,425.778,169.909,33.349,156.294
C06126=1046.846,-38.674,425.764,169.910,33.351,156.294
C06127=1046.852,-38.425,425.751,169.912,33.352,156.295
C06128=1046.858,-38.174,425.738,169.914,33.353,156.295
C06129=1046.864,-37.925,425.725,169.916,33.355,156.295
C06130=1046.871,-37.676,425.712,169.918,33.356,156.295
C06131=1046.877,-37.426,425.699,169.920,33.357,156.295
C06132=1046.883,-37.177,425.686,169.922,33.359,156.295
C06133=1046.889,-36.927,425.673,169.924,33.360,156.295
C06134=1046.896,-36.678,425.659,169.926,33.361,156.296
C06135=1046.902,-36.428,425.646,169.928,33.362,156.296
C06136=1046.908,-36.178,425.633,169.930,33.364,156.296
C06137=1046.914,-35.929,425.620,169.932,33.365,156.296
C06138=1046.920,-35.680,425.607,169.934,33.366,156.296
C06139=1046.927,-35.398,425.592,169.936,33.368,156.296
C06140=1046.934,-35.118,425.577,169.938,33.369,156.297
C06141=1046.942,-34.837,425.562,169.940,33.370,156.297
C06142=1046.948,-34.556,425.547,169.943,33.372,156.297
C06143=1046.954,-34.307,425.534,169.945,33.373,156.297
C06144=1046.961,-34.057,425.520,169.947,33.375,156.297
C06145=1046.967,-33.808,425.507,169.949,33.376,156.298
C06146=1046.973,-33.558,425.494,169.951,33.377,156.298
C06147=1046.979,-33.309,425.481,169.953,33.378,156.298
C06148=1046.986,-33.059,425.467,169.955,33.380,156.298
C06149=1046.992,-32.809,425.454,169.957,33.381,156.298
C06150=1046.998,-32.560,425.441,169.959,33.382,156.298
C06151=1047.005,-32.311,425.428,169.961,33.383,156.298
C06152=1047.011,-32.061,425.414,169.963,33.385,156.299
C06153=1047.018,-31.812,425.401,169.965,33.386,156.299
C06154=1047.023,-31.562,425.387,169.967,33.388,156.299
C06155=1047.030,-31.311,425.374,169.969,33.388,156.299
C06156=1047.036,-31.062,425.361,169.970,33.390,156.299
C06157=1047.042,-30.813,425.347,169.972,33.391,156.299
C06158=1047.048,-30.564,425.334,169.974,33.393,156.300
C06159=1047.055,-30.314,425.320,169.976,33.394,156.300
C06160=1047.061,-30.064,425.307,169.978,33.396,156.300
C06161=1047.067,-29.815,425.294,169.980,33.396,156.300
C06162=1047.074,-29.565,425.280,169.982,33.398,156.300
C06163=1047.080,-29.316,425.266,169.984,33.399,156.300
C06164=1047.086,-29.066,425.253,169.986,33.401,156.301
C06165=1047.093,-28.816,425.240,169.988,33.402,156.301
C06166=1047.099,-28.567,425.226,169.990,33.403,156.301
C06167=1047.106,-28.317,425.213,169.992,33.404,156.301
C06168=1047.112,-28.068,425.199,169.994,33.406,156.301
C06169=1047.118,-27.819,425.186,169.996,33.407,156.302
C06170=1047.124,-27.568,425.172,169.998,33.408,156.302
C06171=1047.131,-27.319,425.159,170.000,33.410,156.302
C06172=1047.137,-27.070,425.145,170.002,33.411,156.302
C06173=1047.144,-26.820,425.132,170.004,33.412,156.302
C06174=1047.150,-26.571,425.118,170.006,33.413,156.302
C06175=1047.155,-26.321,425.105,170.008,33.415,156.303
C06176=1047.162,-26.071,425.091,170.010,33.416,156.303
C06177=1047.168,-25.822,425.078,170.012,33.418,156.303
C06178=1047.175,-25.572,425.063,170.014,33.419,156.303
C06179=1047.181,-25.323,425.049,170.016,33.421,156.303
C06180=1047.186,-25.073,425.036,170.018,33.422,156.303
C06181=1047.193,-24.823,425.022,170.020,33.423,156.304
C06182=1047.199,-24.574,425.009,170.022,33.425,156.304
C06183=1047.205,-24.324,424.995,170.023,33.426,156.304
C06184=1047.212,-24.075,424.981,170.025,33.428,156.304
C06185=1047.218,-23.826,424.967,170.027,33.429,156.304
C06186=1047.224,-23.576,424.953,170.029,33.430,156.305
C06187=1047.230,-23.326,424.940,170.031,33.432,156.305
C06188=1047.236,-23.077,424.926,170.033,33.433,156.305
C06189=1047.243,-22.827,424.912,170.035,33.435,156.305
C06190=1047.249,-22.578,424.898,170.037,33.436,156.305
C06191=1047.255,-22.328,424.884,170.039,33.438,156.306
C06192=1047.262,-22.079,424.871,170.041,33.439,156.306
C06193=1047.268,-21.829,424.857,170.043,33.440,156.306
C06194=1047.274,-21.580,424.842,170.045,33.442,156.306
C06195=1047.280,-21.330,424.829,170.047,33.443,156.306
C06196=1047.286,-21.080,424.815,170.049,33.445,156.307
C06197=1047.293,-20.831,424.802,170.050,33.446,156.307
C06198=1047.300,-20.582,424.787,170.052,33.447,156.307
C06199=1047.305,-20.332,424.773,170.054,33.449,156.307
C06200=1047.312,-20.082,424.760,170.056,33.450,156.307
C06201=1047.318,-19.833,424.745,170.058,33.452,156.307
C06202=1047.325,-19.583,424.732,170.060,33.453,156.308
C06203=1047.332,-19.302,424.716,170.062,33.455,156.308
C06204=1047.338,-19.020,424.701,170.064,33.456,156.308
C06205=1047.346,-18.738,424.685,170.067,33.458,156.308
C06206=1047.353,-18.457,424.669,170.069,33.459,156.309
C06207=1047.359,-18.208,424.656,170.071,33.461,156.309
C06208=1047.365,-17.958,424.641,170.073,33.462,156.309
C06209=1047.372,-17.709,424.628,170.074,33.464,156.309
C06210=1047.378,-17.459,424.613,170.076,33.465,156.309
C06211=1047.384,-17.210,424.599,170.078,33.466,156.310
C06212=1047.390,-16.960,424.585,170.080,33.468,156.310
C06213=1047.397,-16.711,424.571,170.082,33.469,156.310
C06214=1047.404,-16.461,424.557,170.084,33.471,156.310
C06215=1047.410,-16.212,424.543,170.086,33.473,156.310
C06216=1047.416,-15.962,424.529,170.088,33.474,156.311
C06217=1047.422,-15.712,424.515,170.090,33.475,156.311
C06218=1047.429,-15.463,424.501,170.092,33.477,156.311
C06219=1047.435,-15.213,424.487,170.094,33.478,156.311
C06220=1047.441,-14.965,424.473,170.095,33.480,156.311
C06221=1047.447,-14.714,424.459,170.097,33.481,156.312
C06222=1047.454,-14.465,424.444,170.099,33.482,156.312
C06223=1047.460,-14.215,424.430,170.101,33.484,156.312
C06224=1047.466,-13.966,424.415,170.103,33.486,156.312
C06225=1047.472,-13.716,424.402,170.105,33.487,156.312
C06226=1047.479,-13.467,424.387,170.107,33.489,156.313
C06227=1047.484,-13.217,424.373,170.109,33.490,156.313
C06228=1047.491,-12.968,424.358,170.110,33.491,156.313
C06229=1047.497,-12.718,424.345,170.112,33.493,156.313
C06230=1047.503,-12.469,424.330,170.114,33.495,156.313
C06231=1047.509,-12.220,424.316,170.116,33.496,156.314
C06232=1047.516,-11.970,424.302,170.118,33.498,156.314
C06233=1047.522,-11.720,424.287,170.120,33.499,156.314
C06234=1047.528,-11.470,424.273,170.122,33.501,156.314
C06235=1047.535,-11.221,424.259,170.124,33.502,156.314
C06236=1047.541,-10.972,424.244,170.125,33.504,156.315
C06237=1047.547,-10.722,424.230,170.127,33.505,156.315
C06238=1047.554,-10.473,424.216,170.129,33.507,156.315
C06239=1047.559,-10.223,424.202,170.131,33.508,156.315
C06240=1047.566,-9.973,424.187,170.133,33.510,156.316
C06241=1047.572,-9.724,424.172,170.135,33.512,156.316
C06242=1047.578,-9.474,424.159,170.137,33.513,156.316
C06243=1047.585,-9.225,424.144,170.138,33.514,156.316
C06244=1047.591,-8.976,424.129,170.140,33.516,156.316
C06245=1047.597,-8.726,424.115,170.142,33.517,156.317
C06246=1047.603,-8.477,424.101,170.144,33.519,156.317
C06247=1047.610,-8.227,424.086,170.146,33.521,156.317
C06248=1047.616,-7.978,424.071,170.148,33.522,156.317
C06249=1047.622,-7.728,424.058,170.150,33.523,156.318
C06250=1047.629,-7.479,424.043,170.151,33.525,156.318
C06251=1047.635,-7.229,424.028,170.153,33.527,156.318
C06252=1047.641,-6.980,424.015,170.155,33.528,156.318
C06253=1047.648,-6.730,424.000,170.157,33.530,156.318
C06254=1047.654,-6.480,423.985,170.159,33.531,156.319
C06255=1047.660,-6.231,423.970,170.161,33.532,156.319
C06256=1047.667,-5.981,423.956,170.163,33.534,156.319
C06257=1047.673,-5.732,423.941,170.164,33.536,156.319
C06258=1047.679,-5.482,423.927,170.166,33.537,156.319
C06259=1047.685,-5.233,423.912,170.168,33.539,156.320
C06260=1047.692,-4.984,423.898,170.170,33.540,156.320
C06261=1047.698,-4.734,423.883,170.172,33.542,156.320
C06262=1047.704,-4.485,423.869,170.174,33.543,156.320
C06263=1047.711,-4.235,423.854,170.176,33.545,156.321
C06264=1047.718,-3.986,423.840,170.177,33.546,156.321
C06265=1047.724,-3.736,423.825,170.179,33.548,156.321
C06266=1047.730,-3.487,423.810,170.181,33.550,156.321
C06267=1047.737,-3.204,423.794,170.183,33.551,156.321
C06268=1047.744,-2.921,423.777,170.185,33.553,156.322
C06269=1047.751,-2.637,423.760,170.187,33.555,156.322
C06270=1047.759,-2.354,423.743,170.189,33.556,156.322
C06271=1047.764,-2.105,423.728,170.191,33.558,156.323
C06272=1047.770,-1.855,423.713,170.193,33.560,156.323
C06273=1047.776,-1.606,423.698,170.195,33.561,156.323
C06274=1047.782,-1.356,423.684,170.197,33.563,156.323
C06275=1047.788,-1.107,423.669,170.198,33.565,156.323
C06276=1047.795,-0.857,423.654,170.200,33.567,156.324
C06277=1047.800,-0.608,423.640,170.202,33.568,156.324
C06278=1047.807,-0.358,423.625,170.204,33.569,156.324
C06279=1047.813,-0.109,423.610,170.206,33.571,156.324
C06280=1047.820,0.141,423.595,170.207,33.573,156.325
C06281=1047.825,0.390,423.580,170.209,33.575,156.325
C06282=1047.832,0.640,423.565,170.211,33.576,156.325
C06283=1047.838,0.889,423.550,170.213,33.578,156.325
C06284=1047.845,1.139,423.535,170.215,33.580,156.326
C06285=1047.851,1.387,423.520,170.216,33.581,156.326
C06286=1047.857,1.637,423.505,170.218,33.583,156.326
C06287=1047.863,1.887,423.490,170.220,33.584,156.326
C06288=1047.870,2.136,423.475,170.222,33.586,156.327
C06289=1047.875,2.386,423.460,170.224,33.588,156.327
C06290=1047.881,2.635,423.445,170.225,33.589,156.327
C06291=1047.888,2.885,423.430,170.227,33.591,156.327
C06292=1047.894,3.135,423.415,170.229,33.593,156.328
C06293=1047.900,3.384,423.400,170.231,33.594,156.328
C06294=1047.906,3.633,423.386,170.233,33.596,156.328
C06295=1047.913,3.883,423.371,170.234,33.597,156.328
C06296=1047.919,4.132,423.356,170.236,33.599,156.329
C06297=1047.926,4.381,423.340,170.238,33.601,156.329
C06298=1047.932,4.631,423.325,170.240,33.602,156.329
C06299=1047.938,4.880,423.311,170.241,33.604,156.329
C06300=1047.944,5.130,423.296,170.243,33.605,156.330
C06301=1047.950,5.380,423.280,170.245,33.607,156.330
C06302=1047.956,5.629,423.265,170.247,33.609,156.330
C06303=1047.963,5.878,423.250,170.249,33.610,156.330
C06304=1047.969,6.128,423.235,170.250,33.612,156.331
C06305=1047.975,6.377,423.220,170.252,33.614,156.331
C06306=1047.981,6.627,423.205,170.254,33.615,156.331
C06307=1047.988,6.876,423.190,170.256,33.617,156.331
C06308=1047.995,7.125,423.175,170.258,33.618,156.331
C06309=1048.001,7.375,423.160,170.259,33.620,156.332
C06310=1048.007,7.625,423.145,170.261,33.622,156.332
C06311=1048.013,7.875,423.129,170.263,33.623,156.332
C06312=1048.020,8.124,423.113,170.265,33.625,156.332
C06313=1048.026,8.373,423.099,170.266,33.627,156.333
C06314=1048.032,8.622,423.084,170.268,33.629,156.333
C06315=1048.038,8.872,423.069,170.270,33.630,156.333
C06316=1048.045,9.121,423.053,170.272,33.631,156.333
C06317=1048.051,9.371,423.038,170.274,33.633,156.334
C06318=1048.058,9.620,423.023,170.275,33.635,156.334
C06319=1048.064,9.870,423.007,170.278,33.637,156.334
C06320=1048.070,10.119,422.992,170.280,33.638,156.334
C06321=1048.076,10.369,422.977,170.282,33.640,156.335
C06322=1048.083,10.619,422.962,170.283,33.641,156.335
C06323=1048.089,10.868,422.947,170.285,33.643,156.335
C06324=1048.096,11.117,422.932,170.287,33.645,156.335
C06325=1048.102,11.367,422.917,170.289,33.646,156.336
C06326=1048.108,11.616,422.901,170.291,33.648,156.336
C06327=1048.115,11.866,422.886,170.292,33.650,156.336
C06328=1048.121,12.115,422.870,170.294,33.651,156.336
C06329=1048.128,12.365,422.855,170.296,33.653,156.337
C06330=1048.133,12.614,422.840,170.298,33.654,156.337
C06331=1048.141,12.899,422.823,170.300,33.656,156.337
C06332=1048.148,13.184,422.805,170.302,33.658,156.337
C06333=1048.155,13.469,422.788,170.304,33.660,156.338
C06334=1048.163,13.754,422.770,170.306,33.662,156.338
C06335=1048.170,14.003,422.754,170.307,33.663,156.338
C06336=1048.175,14.253,422.739,170.309,33.665,156.338
C06337=1048.182,14.502,422.723,170.311,33.667,156.339
C06338=1048.188,14.751,422.708,170.313,33.669,156.339
C06339=1048.194,15.001,422.693,170.314,33.670,156.339
C06340=1048.201,15.250,422.677,170.316,33.672,156.339
C06341=1048.206,15.500,422.661,170.318,33.673,156.340
C06342=1048.213,15.749,422.646,170.320,33.675,156.340
C06343=1048.220,15.999,422.630,170.321,33.677,156.340
C06344=1048.225,16.248,422.615,170.323,33.679,156.340
C06345=1048.232,16.498,422.599,170.325,33.680,156.341
C06346=1048.238,16.748,422.583,170.327,33.682,156.341
C06347=1048.244,16.997,422.568,170.328,33.684,156.341
C06348=1048.251,17.246,422.553,170.330,33.685,156.342
C06349=1048.257,17.496,422.537,170.332,33.687,156.342
C06350=1048.263,17.745,422.522,170.334,33.689,156.342
C06351=1048.269,17.995,422.505,170.335,33.691,156.342
C06352=1048.276,18.244,422.490,170.337,33.692,156.343
C06353=1048.282,18.493,422.475,170.339,33.694,156.343
C06354=1048.288,18.743,422.458,170.341,33.696,156.343
C06355=1048.294,18.992,422.444,170.342,33.698,156.343
C06356=1048.300,19.242,422.427,170.344,33.699,156.344
C06357=1048.307,19.491,422.412,170.346,33.701,156.344
C06358=1048.313,19.740,422.397,170.347,33.702,156.344
C06359=1048.319,19.990,422.380,170.349,33.704,156.344
C06360=1048.326,20.239,422.365,170.351,33.706,156.345
C06361=1048.332,20.489,422.349,170.353,33.708,156.345
C06362=1048.338,20.738,422.333,170.354,33.710,156.345
C06363=1048.344,20.987,422.317,170.356,33.711,156.345
C06364=1048.350,21.237,422.302,170.358,33.713,156.346
C06365=1048.357,21.486,422.286,170.360,33.714,156.346
C06366=1048.363,21.735,422.270,170.361,33.716,156.346
C06367=1048.369,21.984,422.254,170.363,33.718,156.347
C06368=1048.376,22.235,422.238,170.365,33.720,156.347
C06369=1048.382,22.484,422.223,170.366,33.722,156.347
C06370=1048.388,22.733,422.206,170.368,33.723,156.347
C06371=1048.395,22.983,422.191,170.370,33.725,156.348
C06372=1048.401,23.232,422.175,170.372,33.727,156.348
C06373=1048.407,23.482,422.159,170.374,33.728,156.348
C06374=1048.413,23.731,422.143,170.376,33.730,156.348
C06375=1048.419,23.980,422.127,170.378,33.732,156.349
C06376=1048.426,24.230,422.112,170.379,33.734,156.349
C06377=1048.431,24.479,422.096,170.381,33.736,156.349
C06378=1048.438,24.728,422.080,170.383,33.737,156.349
C06379=1048.445,24.978,422.063,170.385,33.739,156.350
C06380=1048.451,25.228,422.047,170.386,33.740,156.350
C06381=1048.457,25.477,422.032,170.388,33.742,156.350
C06382=1048.463,25.727,422.016,170.390,33.744,156.351
C06383=1048.470,25.976,422.000,170.391,33.746,156.351
C06384=1048.476,26.225,421.984,170.393,33.748,156.351
C06385=1048.482,26.474,421.968,170.395,33.749,156.351
C06386=1048.489,26.724,421.952,170.396,33.751,156.352
C06387=1048.495,26.973,421.936,170.398,33.752,156.352
C06388=1048.502,27.223,421.920,170.400,33.755,156.352
C06389=1048.507,27.472,421.904,170.402,33.757,156.352
C06390=1048.513,27.722,421.888,170.403,33.758,156.353
C06391=1048.520,27.971,421.872,170.405,33.760,156.353
C06392=1048.526,28.221,421.856,170.407,33.762,156.353
C06393=1048.532,28.470,421.840,170.408,33.763,156.354
C06394=1048.539,28.719,421.824,170.410,33.765,156.354
C06395=1048.546,29.006,421.805,170.412,33.767,156.354
C06396=1048.552,29.291,421.786,170.414,33.769,156.354
C06397=1048.560,29.578,421.768,170.416,33.771,156.355
C06398=1048.567,29.865,421.750,170.418,33.773,156.355
C06399=1048.573,30.113,421.733,170.420,33.775,156.355
C06400=1048.579,30.363,421.717,170.421,33.777,156.356
C06401=1048.586,30.612,421.701,170.423,33.779,156.356
C06402=1048.592,30.862,421.684,170.425,33.781,156.356
C06403=1048.598,31.111,421.668,170.426,33.782,156.357
C06404=1048.604,31.360,421.652,170.428,33.784,156.357
C06405=1048.610,31.610,421.636,170.430,33.786,156.357
C06406=1048.618,31.859,421.620,170.431,33.788,156.357
C06407=1048.623,32.109,421.603,170.433,33.789,156.358
C06408=1048.629,32.358,421.587,170.435,33.791,156.358
C06409=1048.635,32.608,421.571,170.436,33.793,156.358
C06410=1048.641,32.857,421.554,170.438,33.794,156.358
C06411=1048.648,33.107,421.538,170.441,33.796,156.359
C06412=1048.655,33.356,421.522,170.442,33.798,156.359
C06413=1048.661,33.605,421.506,170.444,33.800,156.359
C06414=1048.666,33.855,421.490,170.446,33.802,156.360
C06415=1048.673,34.104,421.472,170.447,33.804,156.360
C06416=1048.679,34.353,421.456,170.449,33.806,156.360
C06417=1048.685,34.603,421.440,170.451,33.807,156.360
C06418=1048.692,34.852,421.424,170.453,33.809,156.361
C06419=1048.698,35.102,421.408,170.454,33.811,156.361
C06420=1048.704,35.351,421.391,170.456,33.812,156.361
C06421=1048.711,35.600,421.374,170.458,33.814,156.362
C06422=1048.717,35.849,421.358,170.459,33.816,156.362
C06423=1048.723,36.099,421.341,170.461,33.818,156.362
C06424=1048.730,36.348,421.326,170.463,33.820,156.362
C06425=1048.736,36.598,421.310,170.464,33.822,156.363
C06426=1048.742,36.847,421.293,170.466,33.823,156.363
C06427=1048.749,37.096,421.276,170.468,33.825,156.363
C06428=1048.755,37.346,421.260,170.469,33.827,156.364
C06429=1048.761,37.595,421.243,170.471,33.828,156.364
C06430=1048.767,37.845,421.227,170.473,33.830,156.364
C06431=1048.773,38.094,421.210,170.474,33.832,156.364
C06432=1048.779,38.343,421.194,170.476,33.834,156.365
C06433=1048.785,38.593,421.177,170.478,33.836,156.365
C06434=1048.792,38.842,421.160,170.479,33.838,156.365
C06435=1048.798,39.091,421.144,170.481,33.840,156.366
C06436=1048.804,39.341,421.127,170.483,33.842,156.366
C06437=1048.811,39.591,421.111,170.484,33.843,156.366
C06438=1048.817,39.840,421.094,170.486,33.845,156.366
C06439=1048.823,40.089,421.078,170.488,33.847,156.367
C06440=1048.829,40.338,421.061,170.489,33.849,156.367
C06441=1048.836,40.588,421.044,170.491,33.851,156.367
C06442=1048.842,40.837,421.028,170.494,33.852,156.368
C06443=1048.848,41.086,421.011,170.495,33.854,156.368
C06444=1048.854,41.336,420.994,170.497,33.856,156.368
C06445=1048.860,41.585,420.978,170.499,33.858,156.369
C06446=1048.866,41.834,420.960,170.500,33.859,156.369
C06447=1048.872,42.084,420.944,170.502,33.861,156.369
C06448=1048.878,42.334,420.927,170.504,33.863,156.369
C06449=1048.885,42.582,420.910,170.505,33.865,156.370
C06450=1048.891,42.832,420.894,170.507,33.867,156.370
C06451=1048.897,43.081,420.877,170.508,33.869,156.370
C06452=1048.904,43.331,420.860,170.510,33.871,156.371
C06453=1048.910,43.580,420.843,170.512,33.873,156.371
C06454=1048.916,43.829,420.827,170.513,33.875,156.371
C06455=1048.922,44.078,420.809,170.515,33.877,156.372
C06456=1048.928,44.328,420.793,170.517,33.879,156.372
C06457=1048.934,44.577,420.776,170.518,33.880,156.372
C06458=1048.940,44.827,420.759,170.520,33.882,156.372
C06459=1048.947,45.112,420.740,170.522,33.884,156.373
C06460=1048.955,45.400,420.720,170.524,33.886,156.373
C06461=1048.962,45.686,420.700,170.526,33.888,156.373
C06462=1048.968,45.972,420.681,170.527,33.891,156.374
C06463=1048.975,46.221,420.664,170.529,33.892,156.374
C06464=1048.980,46.470,420.648,170.531,33.894,156.374
C06465=1048.987,46.720,420.630,170.532,33.896,156.375
C06466=1048.993,46.969,420.613,170.534,33.898,156.375
C06467=1048.999,47.218,420.597,170.537,33.900,156.375
C06468=1049.005,47.468,420.579,170.538,33.902,156.376
C06469=1049.011,47.717,420.562,170.540,33.904,156.376
C06470=1049.018,47.967,420.545,170.542,33.906,156.376
C06471=1049.023,48.216,420.528,170.543,33.907,156.376
C06472=1049.029,48.465,420.511,170.545,33.909,156.377
C06473=1049.036,48.714,420.494,170.546,33.911,156.377
C06474=1049.041,48.964,420.477,170.548,33.913,156.377
C06475=1049.048,49.213,420.460,170.550,33.915,156.378
C06476=1049.054,49.463,420.443,170.551,33.917,156.378
C06477=1049.060,49.712,420.426,170.553,33.919,156.378
C06478=1049.066,49.961,420.408,170.555,33.921,156.379
C06479=1049.072,50.211,420.392,170.556,33.923,156.379
C06480=1049.079,50.460,420.374,170.558,33.925,156.379
C06481=1049.085,50.709,420.357,170.560,33.927,156.380
C06482=1049.092,50.958,420.340,170.561,33.928,156.380
C06483=1049.097,51.208,420.323,170.563,33.930,156.380
C06484=1049.103,51.457,420.306,170.564,33.932,156.381
C06485=1049.110,51.706,420.289,170.566,33.934,156.381
C06486=1049.115,51.956,420.272,170.568,33.936,156.381
C06487=1049.122,52.205,420.255,170.569,33.938,156.381
C06488=1049.128,52.454,420.237,170.571,33.940,156.382
C06489=1049.134,52.704,420.220,170.573,33.942,156.382
C06490=1049.140,52.953,420.203,170.574,33.944,156.382
C06491=1049.147,53.203,420.186,170.577,33.946,156.383
C06492=1049.153,53.452,420.169,170.579,33.948,156.383
C06493=1049.160,53.701,420.151,170.580,33.949,156.383
C06494=1049.165,53.950,420.134,170.582,33.951,156.384
C06495=1049.172,54.200,420.117,170.583,33.953,156.384
C06496=1049.177,54.449,420.099,170.585,33.955,156.384
C06497=1049.184,54.699,420.082,170.587,33.957,156.384
C06498=1049.190,54.947,420.065,170.588,33.959,156.385
C06499=1049.196,55.197,420.047,170.590,33.960,156.385
C06500=1049.202,55.446,420.031,170.592,33.962,156.385
C06501=1049.209,55.696,420.013,170.593,33.964,156.386
C06502=1049.215,55.945,419.996,170.595,33.966,156.386
C06503=1049.222,56.194,419.979,170.597,33.968,156.386
C06504=1049.227,56.443,419.961,170.598,33.970,156.387
C06505=1049.234,56.693,419.944,170.600,33.971,156.387
C06506=1049.241,56.942,419.926,170.601,33.973,156.387
C06507=1049.246,57.192,419.910,170.603,33.975,156.387
C06508=1049.253,57.441,419.892,170.605,33.977,156.388
C06509=1049.258,57.690,419.875,170.606,33.979,156.388
C06510=1049.265,57.940,419.857,170.608,33.981,156.388
C06511=1049.271,58.189,419.840,170.610,33.982,156.389
C06512=1049.278,58.438,419.822,170.611,33.984,156.389
C06513=1049.285,58.688,419.805,170.613,33.986,156.389
C06514=1049.290,58.937,419.788,170.616,33.988,156.390
C06515=1049.297,59.186,419.770,170.617,33.990,156.390
C06516=1049.302,59.435,419.753,170.619,33.991,156.390
C06517=1049.309,59.685,419.735,170.620,33.993,156.390
C06518=1049.316,59.934,419.718,170.622,33.995,156.391
C06519=1049.322,60.183,419.700,170.624,33.997,156.391
C06520=1049.329,60.433,419.683,170.625,33.999,156.391
C06521=1049.334,60.682,419.666,170.627,34.001,156.392
C06522=1049.341,60.931,419.648,170.629,34.003,156.392
C06523=1049.348,61.217,419.628,170.631,34.005,156.392
C06524=1049.355,61.503,419.608,170.632,34.007,156.393
C06525=1049.362,61.790,419.588,170.634,34.009,156.393
C06526=1049.370,62.075,419.569,170.636,34.011,156.393
C06527=1049.376,62.325,419.551,170.638,34.013,156.394
C06528=1049.382,62.574,419.534,170.640,34.015,156.394
C06529=1049.389,62.823,419.515,170.641,34.016,156.394
C06530=1049.396,63.072,419.498,170.643,34.018,156.395
C06531=1049.401,63.321,419.480,170.644,34.020,156.395
C06532=1049.408,63.571,419.463,170.646,34.022,156.395
C06533=1049.414,63.820,419.445,170.648,34.024,156.396
C06534=1049.421,64.069,419.428,170.649,34.026,156.396
C06535=1049.427,64.319,419.410,170.652,34.028,156.396
C06536=1049.434,64.568,419.393,170.654,34.030,156.396
C06537=1049.439,64.817,419.375,170.655,34.031,156.397
C06538=1049.445,65.067,419.357,170.657,34.033,156.397
C06539=1049.452,65.316,419.338,170.659,34.035,156.397
C06540=1049.458,65.565,419.321,170.660,34.037,156.398
C06541=1049.464,65.815,419.304,170.662,34.039,156.398
C06542=1049.470,66.064,419.286,170.663,34.041,156.398
C06543=1049.476,66.313,419.269,170.665,34.043,156.399
C06544=1049.483,66.562,419.250,170.667,34.045,156.399
C06545=1049.489,66.812,419.232,170.668,34.047,156.399
C06546=1049.495,67.061,419.215,170.670,34.048,156.399
C06547=1049.501,67.310,419.197,170.672,34.050,156.400
C06548=1049.507,67.560,419.179,170.673,34.052,156.400
C06549=1049.513,67.809,419.161,170.675,34.054,156.400
C06550=1049.520,68.058,419.144,170.676,34.056,156.401
C06551=1049.527,68.328,419.124,170.678,34.058,156.401
C06552=1049.533,68.596,419.105,170.680,34.060,156.401
C06553=1049.540,68.866,419.085,170.682,34.063,156.402
C06554=1049.547,69.134,419.067,170.684,34.065,156.402
C06555=1049.553,69.384,419.049,170.686,34.067,156.403
C06556=1049.559,69.633,419.030,170.688,34.069,156.403
C06557=1049.565,69.883,419.012,170.689,34.071,156.403
C06558=1049.571,70.132,418.995,170.691,34.073,156.403
C06559=1049.577,70.381,418.976,170.692,34.074,156.404
C06560=1049.584,70.630,418.959,170.694,34.076,156.404
C06561=1049.590,70.879,418.941,170.696,34.078,156.404
C06562=1049.596,71.129,418.922,170.697,34.080,156.405
C06563=1049.602,71.378,418.904,170.699,34.082,156.405
C06564=1049.608,71.628,418.886,170.701,34.084,156.405
C06565=1049.614,71.876,418.868,170.702,34.086,156.406
C06566=1049.620,72.126,418.850,170.704,34.087,156.406
C06567=1049.627,72.375,418.832,170.705,34.089,156.406
C06568=1049.632,72.624,418.814,170.707,34.091,156.407
C06569=1049.638,72.873,418.795,170.709,34.093,156.407
C06570=1049.645,73.123,418.778,170.710,34.095,156.407
C06571=1049.651,73.373,418.760,170.712,34.097,156.408
C06572=1049.657,73.621,418.742,170.714,34.099,156.408
C06573=1049.663,73.871,418.724,170.716,34.101,156.408
C06574=1049.670,74.120,418.705,170.718,34.103,156.409
C06575=1049.676,74.370,418.687,170.719,34.105,156.409
C06576=1049.682,74.618,418.669,170.721,34.107,156.409
C06577=1049.688,74.868,418.651,170.723,34.109,156.410
C06578=1049.694,75.117,418.632,170.724,34.111,156.410
C06579=1049.700,75.367,418.615,170.726,34.113,156.410
C06580=1049.707,75.616,418.596,170.727,34.115,156.411
C06581=1049.712,75.865,418.578,170.729,34.117,156.411
C06582=1049.719,76.114,418.560,170.731,34.119,156.411
C06583=1049.725,76.364,418.542,170.732,34.121,156.412
C06584=1049.731,76.613,418.523,170.734,34.123,156.412
C06585=1049.738,76.862,418.506,170.736,34.125,156.412
C06586=1049.744,77.111,418.487,170.737,34.126,156.412
C06587=1049.751,77.377,418.468,170.739,34.128,156.413
C06588=1049.757,77.643,418.448,170.741,34.130,156.413
C06589=1049.764,77.910,418.428,170.743,34.132,156.413
C06590=1049.771,78.174,418.409,170.745,34.134,156.414
C06591=1049.777,78.424,418.391,170.747,34.136,156.414
C06592=1049.783,78.673,418.373,170.748,34.138,156.414
C06593=1049.788,78.923,418.354,170.750,34.141,156.415
C06594=1049.794,79.172,418.335,170.752,34.143,156.415
C06595=1049.801,79.421,418.317,170.753,34.145,156.416
C06596=1049.807,79.671,418.299,170.755,34.147,156.416
C06597=1049.813,79.920,418.280,170.756,34.148,156.416
C06598=1049.819,80.169,418.261,170.758,34.150,156.417
C06599=1049.825,80.418,418.243,170.760,34.152,156.417
C06600=1049.831,80.667,418.225,170.761,34.154,156.417
C06601=1049.837,80.917,418.206,170.763,34.156,156.417
C06602=1049.844,81.166,418.187,170.764,34.158,156.418
C06603=1049.849,81.415,418.170,170.766,34.160,156.418
C06604=1049.855,81.664,418.151,170.768,34.162,156.418
C06605=1049.862,81.913,418.132,170.770,34.164,156.419
C06606=1049.868,82.162,418.113,170.772,34.166,156.419
C06607=1049.874,82.412,418.095,170.774,34.168,156.419
C06608=1049.881,82.661,418.077,170.775,34.170,156.420
C06609=1049.886,82.911,418.057,170.777,34.172,156.420
C06610=1049.892,83.159,418.039,170.778,34.174,156.420
C06611=1049.898,83.409,418.021,170.780,34.176,156.421
C06612=1049.905,83.658,418.003,170.782,34.178,156.421
C06613=1049.910,83.907,417.983,170.783,34.180,156.422
C06614=1049.917,84.156,417.965,170.785,34.182,156.422
C06615=1049.923,84.406,417.946,170.787,34.184,156.422
C06616=1049.929,84.655,417.928,170.788,34.186,156.423
C06617=1049.936,84.904,417.909,170.790,34.188,156.423
C06618=1049.941,85.154,417.890,170.791,34.190,156.423
C06619=1049.947,85.402,417.872,170.793,34.192,156.423
C06620=1049.954,85.651,417.853,170.795,34.194,156.424
C06621=1049.960,85.901,417.835,170.797,34.196,156.424
C06622=1049.966,86.150,417.815,170.799,34.198,156.424
C06623=1049.972,86.400,417.797,170.801,34.200,156.425
C06624=1049.978,86.649,417.779,170.802,34.202,156.425
C06625=1049.985,86.898,417.760,170.804,34.204,156.425
C06626=1049.990,87.147,417.741,170.805,34.205,156.426
C06627=1049.997,87.397,417.722,170.807,34.207,156.426
C06628=1050.003,87.646,417.704,170.809,34.209,156.426
C06629=1050.010,87.895,417.685,170.810,34.211,156.427
C06630=1050.015,88.144,417.666,170.812,34.213,156.427
C06631=1050.022,88.393,417.647,170.814,34.215,156.427
C06632=1050.028,88.642,417.628,170.815,34.217,156.428
C06633=1050.035,88.892,417.610,170.817,34.219,156.428
C06634=1050.040,89.141,417.591,170.818,34.221,156.428
C06635=1050.047,89.390,417.572,170.820,34.223,156.429
C06636=1050.053,89.640,417.554,170.823,34.225,156.429
C06637=1050.059,89.889,417.535,170.824,34.227,156.429
C06638=1050.065,90.138,417.516,170.826,34.229,156.430
C06639=1050.071,90.388,417.497,170.828,34.231,156.430
C06640=1050.078,90.637,417.479,170.829,34.233,156.430
C06641=1050.084,90.885,417.459,170.831,34.235,156.431
C06642=1050.090,91.135,417.440,170.833,34.237,156.431
C06643=1050.096,91.384,417.421,170.834,34.238,156.431
C06644=1050.102,91.633,417.402,170.836,34.240,156.432
C06645=1050.108,91.883,417.383,170.837,34.243,156.432
C06646=1050.114,92.132,417.364,170.839,34.245,156.432
C06647=1050.120,92.381,417.345,170.841,34.247,156.433
C06648=1050.127,92.630,417.326,170.842,34.249,156.433
C06649=1050.132,92.879,417.308,170.844,34.251,156.433
C06650=1050.138,93.128,417.289,170.846,34.253,156.434
C06651=1050.146,93.414,417.267,170.848,34.255,156.434
C06652=1050.153,93.700,417.245,170.850,34.257,156.435
C06653=1050.159,93.985,417.222,170.852,34.260,156.435
C06654=1050.166,94.272,417.201,170.854,34.262,156.435
C06655=1050.173,94.520,417.181,170.856,34.264,156.436
C06656=1050.178,94.770,417.162,170.857,34.266,156.436
C06657=1050.185,95.019,417.144,170.859,34.268,156.436
C06658=1050.190,95.268,417.124,170.861,34.270,156.437
C06659=1050.197,95.517,417.106,170.862,34.272,156.437
C06660=1050.203,95.766,417.086,170.864,34.274,156.437
C06661=1050.209,96.015,417.067,170.865,34.276,156.438
C06662=1050.215,96.265,417.048,170.867,34.278,156.438
C06663=1050.221,96.514,417.029,170.869,34.280,156.438
C06664=1050.227,96.763,417.010,170.871,34.282,156.439
C06665=1050.234,97.012,416.991,170.873,34.284,156.439
C06666=1050.240,97.261,416.971,170.875,34.285,156.439
C06667=1050.245,97.511,416.952,170.876,34.287,156.440
C06668=1050.252,97.760,416.933,170.878,34.290,156.440
C06669=1050.258,98.009,416.913,170.880,34.292,156.440
C06670=1050.264,98.258,416.895,170.881,34.294,156.441
C06671=1050.270,98.508,416.875,170.883,34.296,156.441
C06672=1050.277,98.756,416.856,170.884,34.298,156.441
C06673=1050.283,99.006,416.837,170.886,34.300,156.442
C06674=1050.289,99.255,416.818,170.888,34.302,156.442
C06675=1050.295,99.504,416.798,170.889,34.303,156.442
C06676=1050.301,99.753,416.779,170.891,34.305,156.443
C06677=1050.307,100.002,416.760,170.893,34.307,156.443
C06678=1050.313,100.251,416.740,170.895,34.309,156.443
C06679=1050.320,100.500,416.721,170.897,34.311,156.444
C06680=1050.326,100.750,416.702,170.899,34.313,156.444
C06681=1050.332,100.999,416.682,170.900,34.316,156.445
C06682=1050.338,101.249,416.663,170.902,34.318,156.445
C06683=1050.344,101.497,416.643,170.904,34.320,156.445
C06684=1050.350,101.747,416.624,170.905,34.321,156.446
C06685=1050.356,101.996,416.605,170.907,34.323,156.446
C06686=1050.362,102.245,416.585,170.909,34.325,156.446
C06687=1050.367,102.494,416.566,170.910,34.328,156.447
C06688=1050.374,102.743,416.546,170.912,34.330,156.447
C06689=1050.380,102.993,416.527,170.913,34.332,156.447
C06690=1050.386,103.242,416.507,170.915,34.334,156.448
C06691=1050.392,103.491,416.487,170.918,34.336,156.448
C06692=1050.398,103.740,416.467,170.919,34.338,156.448
C06693=1050.405,103.989,416.449,170.921,34.340,156.449
C06694=1050.411,104.238,416.429,170.923,34.342,156.449
C06695=1050.416,104.487,416.410,170.924,34.344,156.449
C06696=1050.422,104.736,416.390,170.926,34.346,156.450
C06697=1050.429,104.986,416.370,170.928,34.348,156.450
C06698=1050.435,105.235,416.350,170.929,34.350,156.450
C06699=1050.441,105.484,416.331,170.931,34.352,156.451
C06700=1050.447,105.733,416.311,170.933,34.354,156.451
C06701=1050.453,105.982,416.292,170.934,34.356,156.452
C06702=1050.459,106.231,416.272,170.936,34.358,156.452
C06703=1050.465,106.481,416.252,170.939,34.360,156.452
C06704=1050.471,106.730,416.233,170.940,34.362,156.453
C06705=1050.478,106.979,416.213,170.942,34.364,156.453
C06706=1050.483,107.228,416.194,170.944,34.366,156.453
C06707=1050.489,107.477,416.174,170.945,34.368,156.454
C06708=1050.496,107.726,416.154,170.947,34.370,156.454
C06709=1050.502,107.976,416.135,170.949,34.372,156.454
C06710=1050.508,108.225,416.115,170.950,34.374,156.455
C06711=1050.514,108.473,416.095,170.952,34.376,156.455
C06712=1050.521,108.723,416.076,170.954,34.378,156.455
C06713=1050.527,108.972,416.056,170.955,34.381,156.456
C06714=1050.532,109.222,416.036,170.957,34.382,156.456
C06715=1050.540,109.507,416.013,170.959,34.384,156.456
C06716=1050.547,109.793,415.990,170.962,34.387,156.457
C06717=1050.554,110.078,415.968,170.964,34.389,156.457
C06718=1050.560,110.364,415.946,170.966,34.391,156.458
C06719=1050.567,110.613,415.925,170.967,34.393,156.458
C06720=1050.573,110.863,415.906,170.969,34.395,156.458
C06721=1050.579,111.111,415.886,170.971,34.397,156.459
C06722=1050.585,111.360,415.866,170.972,34.400,156.459
C06723=1050.591,111.610,415.846,170.974,34.402,156.459
C06724=1050.597,111.859,415.826,170.976,34.404,156.460
C06725=1050.603,112.108,415.806,170.977,34.406,156.460
C06726=1050.609,112.357,415.787,170.979,34.407,156.460
C06727=1050.615,112.606,415.766,170.982,34.410,156.461
C06728=1050.621,112.855,415.746,170.983,34.412,156.461
C06729=1050.627,113.105,415.727,170.985,34.414,156.461
C06730=1050.634,113.354,415.707,170.987,34.416,156.462
C06731=1050.640,113.603,415.687,170.988,34.418,156.462
C06732=1050.646,113.852,415.667,170.990,34.420,156.463
C06733=1050.652,114.101,415.647,170.992,34.422,156.463
C06734=1050.658,114.350,415.626,170.993,34.424,156.463
C06735=1050.664,114.599,415.606,170.995,34.426,156.464
C06736=1050.669,114.849,415.587,170.997,34.429,156.464
C06737=1050.675,115.097,415.567,170.998,34.430,156.464
C06738=1050.682,115.347,415.546,171.000,34.432,156.465
C06739=1050.687,115.596,415.526,171.003,34.435,156.465
C06740=1050.693,115.845,415.506,171.004,34.437,156.466
C06741=1050.699,116.094,415.486,171.006,34.439,156.466
C06742=1050.706,116.343,415.466,171.008,34.441,156.466
C06743=1050.711,116.592,415.445,171.009,34.443,156.467
C06744=1050.717,116.841,415.425,171.011,34.445,156.467
C06745=1050.724,117.091,415.405,171.013,34.447,156.467
C06746=1050.730,117.339,415.385,171.014,34.450,156.468
C06747=1050.735,117.589,415.364,171.016,34.452,156.468
C06748=1050.741,117.837,415.344,171.018,34.453,156.468
C06749=1050.747,118.087,415.324,171.020,34.456,156.469
C06750=1050.753,118.336,415.303,171.022,34.458,156.469
C06751=1050.759,118.585,415.283,171.024,34.460,156.470
C06752=1050.765,118.834,415.263,171.025,34.462,156.470
C06753=1050.771,119.083,415.243,171.027,34.464,156.470
C06754=1050.776,119.332,415.223,171.029,34.466,156.471
C06755=1050.783,119.582,415.202,171.031,34.468,156.471
C06756=1050.789,119.831,415.182,171.032,34.471,156.471
C06757=1050.794,120.080,415.162,171.034,34.473,156.472
C06758=1050.801,120.329,415.141,171.036,34.475,156.472
C06759=1050.807,120.577,415.121,171.037,34.476,156.472
C06760=1050.813,120.826,415.101,171.040,34.479,156.473
C06761=1050.819,121.076,415.080,171.042,34.481,156.473
C06762=1050.825,121.325,415.060,171.043,34.483,156.474
C06763=1050.832,121.574,415.040,171.045,34.485,156.474
C06764=1050.837,121.824,415.019,171.047,34.487,156.474
C06765=1050.843,122.072,414.999,171.049,34.489,156.475
C06766=1050.849,122.322,414.979,171.050,34.491,156.475
C06767=1050.855,122.570,414.958,171.052,34.493,156.475
C06768=1050.862,122.820,414.937,171.054,34.496,156.476
C06769=1050.868,123.069,414.917,171.055,34.497,156.476
C06770=1050.873,123.318,414.897,171.057,34.499,156.476
C06771=1050.879,123.567,414.876,171.060,34.501,156.477
C06772=1050.886,123.816,414.856,171.062,34.504,156.477
C06773=1050.892,124.065,414.835,171.063,34.506,156.478
C06774=1050.898,124.314,414.815,171.065,34.508,156.478
C06775=1050.904,124.563,414.795,171.067,34.510,156.478
C06776=1050.909,124.813,414.774,171.068,34.512,156.479
C06777=1050.916,125.061,414.753,171.070,34.514,156.479
C06778=1050.922,125.311,414.733,171.072,34.516,156.479
C06779=1050.929,125.596,414.709,171.074,34.519,156.480
C06780=1050.936,125.882,414.686,171.076,34.521,156.480
C06781=1050.943,126.167,414.663,171.078,34.523,156.481
C06782=1050.950,126.453,414.639,171.081,34.526,156.481
C06783=1050.957,126.702,414.619,171.082,34.527,156.481
C06784=1050.962,126.951,414.597,171.084,34.530,156.482
C06785=1050.969,127.200,414.577,171.086,34.532,156.482
C06786=1050.974,127.449,414.557,171.088,34.534,156.482
C06787=1050.981,127.698,414.536,171.089,34.536,156.483
C06788=1050.987,127.947,414.516,171.091,34.538,156.483
C06789=1050.993,128.197,414.495,171.093,34.540,156.484
C06790=1050.999,128.445,414.474,171.095,34.542,156.484
C06791=1051.006,128.695,414.454,171.096,34.544,156.484
C06792=1051.011,128.944,414.433,171.099,34.546,156.485
C06793=1051.018,129.193,414.412,171.101,34.548,156.485
C06794=1051.024,129.441,414.392,171.103,34.550,156.485
C06795=1051.030,129.691,414.370,171.104,34.552,156.486
C06796=1051.036,129.939,414.350,171.106,34.554,156.486
C06797=1051.042,130.189,414.330,171.108,34.556,156.486
C06798=1051.048,130.437,414.309,171.110,34.559,156.487
C06799=1051.055,130.687,414.289,171.111,34.561,156.487
C06800=1051.061,130.936,414.267,171.113,34.563,156.487
C06801=1051.067,131.185,414.247,171.115,34.564,156.488
C06802=1051.074,131.434,414.226,171.118,34.566,156.488
C06803=1051.079,131.683,414.205,171.119,34.569,156.489
C06804=1051.085,131.932,414.184,171.121,34.571,156.489
C06805=1051.091,132.181,414.164,171.123,34.573,156.489
C06806=1051.097,132.430,414.142,171.125,34.575,156.490
C06807=1051.103,132.679,414.122,171.126,34.577,156.490
C06808=1051.110,132.928,414.101,171.128,34.580,156.491
C06809=1051.115,133.177,414.080,171.130,34.582,156.491
C06810=1051.121,133.427,414.058,171.132,34.584,156.491
C06811=1051.128,133.676,414.038,171.133,34.586,156.492
C06812=1051.133,133.925,414.017,171.136,34.588,156.492
C06813=1051.139,134.174,413.995,171.138,34.590,156.492
C06814=1051.145,134.423,413.975,171.140,34.592,156.493
C06815=1051.151,134.672,413.954,171.142,34.594,156.493
C06816=1051.157,134.921,413.933,171.143,34.596,156.493
C06817=1051.164,135.170,413.912,171.145,34.599,156.494
C06818=1051.170,135.419,413.890,171.147,34.601,156.494
C06819=1051.175,135.668,413.870,171.149,34.603,156.495
C06820=1051.182,135.917,413.849,171.150,34.605,156.495
C06821=1051.188,136.166,413.827,171.152,34.607,156.495
C06822=1051.193,136.415,413.807,171.155,34.609,156.496
C06823=1051.200,136.665,413.785,171.157,34.611,156.496
C06824=1051.206,136.913,413.764,171.158,34.613,156.496
C06825=1051.212,137.163,413.743,171.160,34.616,156.497
C06826=1051.217,137.411,413.722,171.162,34.618,156.497
C06827=1051.224,137.660,413.701,171.164,34.620,156.498
C06828=1051.230,137.910,413.680,171.166,34.622,156.498
C06829=1051.236,138.158,413.659,171.167,34.624,156.498
C06830=1051.242,138.408,413.637,171.169,34.626,156.499
C06831=1051.248,138.656,413.616,171.172,34.629,156.499
C06832=1051.254,138.906,413.596,171.174,34.631,156.500
C06833=1051.260,139.155,413.574,171.175,34.632,156.500
C06834=1051.266,139.403,413.553,171.177,34.635,156.500
C06835=1051.273,139.652,413.532,171.179,34.637,156.501
C06836=1051.279,139.901,413.510,171.181,34.639,156.501
C06837=1051.284,140.151,413.489,171.183,34.641,156.501
C06838=1051.290,140.400,413.468,171.184,34.643,156.502
C06839=1051.296,140.649,413.446,171.186,34.646,156.502
C06840=1051.302,140.897,413.425,171.188,34.648,156.503
C06841=1051.308,141.147,413.403,171.191,34.650,156.503
C06842=1051.314,141.396,413.382,171.193,34.652,156.503
C06843=1051.321,141.681,413.358,171.195,34.655,156.504
C06844=1051.328,141.966,413.333,171.197,34.657,156.504
C06845=1051.334,142.252,413.309,171.199,34.660,156.505
C06846=1051.341,142.537,413.284,171.201,34.662,156.505
C06847=1051.347,142.786,413.263,171.203,34.664,156.506
C06848=1051.354,143.035,413.241,171.204,34.667,156.506
C06849=1051.359,143.284,413.220,171.207,34.669,156.506
C06850=1051.365,143.533,413.198,171.209,34.671,156.507
C06851=1051.372,143.782,413.177,171.211,34.673,156.507
C06852=1051.377,144.031,413.155,171.213,34.675,156.507
C06853=1051.383,144.280,413.134,171.214,34.677,156.508
C06854=1051.389,144.529,413.112,171.216,34.679,156.508
C06855=1051.396,144.778,413.090,171.218,34.682,156.509
C06856=1051.401,145.027,413.069,171.220,34.684,156.509
C06857=1051.407,145.276,413.047,171.222,34.686,156.509
C06858=1051.413,145.525,413.026,171.224,34.688,156.510
C06859=1051.420,145.774,413.005,171.226,34.690,156.510
C06860=1051.426,146.023,412.984,171.228,34.693,156.511
C06861=1051.432,146.272,412.962,171.230,34.694,156.511
C06862=1051.438,146.521,412.940,171.232,34.697,156.511
C06863=1051.444,146.770,412.919,171.234,34.699,156.512
C06864=1051.450,147.019,412.897,171.235,34.701,156.512
C06865=1051.456,147.268,412.876,171.237,34.703,156.513
C06866=1051.462,147.517,412.854,171.239,34.705,156.513
C06867=1051.468,147.766,412.832,171.242,34.708,156.513
C06868=1051.474,148.015,412.811,171.244,34.710,156.514
C06869=1051.479,148.264,412.789,171.246,34.712,156.514
C06870=1051.486,148.513,412.767,171.247,34.714,156.514
C06871=1051.492,148.762,412.745,171.249,34.717,156.515
C06872=1051.498,149.011,412.724,171.251,34.718,156.515
C06873=1051.504,149.260,412.702,171.253,34.721,156.516
C06874=1051.510,149.509,412.680,171.255,34.723,156.516
C06875=1051.516,149.758,412.659,171.258,34.725,156.516
C06876=1051.523,150.007,412.636,171.259,34.727,156.517
C06877=1051.527,150.256,412.615,171.261,34.730,156.517
C06878=1051.534,150.505,412.593,171.263,34.732,156.518
C06879=1051.540,150.754,412.571,171.265,34.734,156.518
C06880=1051.546,151.003,412.549,171.267,34.736,156.518
C06881=1051.552,151.252,412.527,171.269,34.739,156.519
C06882=1051.557,151.501,412.505,171.271,34.741,156.519
C06883=1051.563,151.750,412.484,171.273,34.743,156.520
C06884=1051.570,151.998,412.461,171.275,34.746,156.520
C06885=1051.576,152.248,412.440,171.277,34.748,156.520
C06886=1051.582,152.497,412.418,171.279,34.750,156.521
C06887=1051.587,152.745,412.396,171.281,34.752,156.521
C06888=1051.593,152.994,412.374,171.283,34.754,156.522
C06889=1051.600,153.243,412.352,171.285,34.756,156.522
C06890=1051.606,153.492,412.330,171.286,34.759,156.523
C06891=1051.612,153.742,412.308,171.288,34.761,156.523
C06892=1051.618,153.991,412.286,171.291,34.763,156.523
C06893=1051.624,154.239,412.264,171.293,34.765,156.524
C06894=1051.630,154.488,412.243,171.295,34.768,156.524
C06895=1051.636,154.737,412.221,171.297,34.770,156.524
C06896=1051.642,154.986,412.198,171.299,34.772,156.525
C06897=1051.648,155.235,412.176,171.301,34.774,156.525
C06898=1051.654,155.484,412.154,171.302,34.777,156.526
C06899=1051.660,155.733,412.132,171.305,34.779,156.526
C06900=1051.666,155.983,412.110,171.307,34.781,156.526
C06901=1051.672,156.231,412.088,171.309,34.783,156.527
C06902=1051.677,156.480,412.066,171.311,34.785,156.527
C06903=1051.684,156.728,412.044,171.313,34.788,156.528
C06904=1051.689,156.978,412.021,171.315,34.790,156.528
C06905=1051.696,157.227,411.999,171.317,34.792,156.529
C06906=1051.702,157.476,411.977,171.318,34.795,156.529
C06907=1051.709,157.760,411.952,171.322,34.797,156.529
C06908=1051.716,158.046,411.926,171.324,34.800,156.530
C06909=1051.723,158.330,411.901,171.326,34.802,156.530
C06910=1051.729,158.616,411.876,171.328,34.805,156.531
C06911=1051.735,158.864,411.853,171.330,34.807,156.531
C06912=1051.741,159.114,411.831,171.332,34.809,156.532
C06913=1051.747,159.363,411.808,171.334,34.812,156.532
C06914=1051.753,159.612,411.786,171.336,34.814,156.532
C06915=1051.759,159.860,411.764,171.339,34.816,156.533
C06916=1051.765,160.110,411.742,171.341,34.819,156.533
C06917=1051.771,160.358,411.720,171.343,34.821,156.534
C06918=1051.777,160.607,411.697,171.344,34.823,156.534
C06919=1051.783,160.857,411.675,171.346,34.825,156.534
C06920=1051.789,161.105,411.652,171.348,34.828,156.535
C06921=1051.795,161.354,411.629,171.350,34.830,156.535
C06922=1051.801,161.604,411.607,171.353,34.833,156.536
C06923=1051.807,161.852,411.584,171.355,34.835,156.536
C06924=1051.812,162.101,411.562,171.357,34.837,156.537
C06925=1051.817,162.350,411.539,171.359,34.839,156.537
C06926=1051.824,162.599,411.517,171.361,34.842,156.538
C06927=1051.829,162.848,411.494,171.362,34.844,156.538
C06928=1051.835,163.097,411.471,171.364,34.847,156.538
C06929=1051.841,163.345,411.448,171.367,34.849,156.539
C06930=1051.847,163.595,411.427,171.369,34.851,156.539
C06931=1051.853,163.844,411.404,171.371,34.854,156.540
C06932=1051.858,164.092,411.381,171.373,34.856,156.540
C06933=1051.864,164.341,411.358,171.375,34.858,156.541
C06934=1051.870,164.590,411.335,171.377,34.861,156.541
C06935=1051.876,164.839,411.313,171.379,34.863,156.541
C06936=1051.882,165.088,411.290,171.382,34.866,156.542
C06937=1051.888,165.337,411.268,171.384,34.868,156.542
C06938=1051.893,165.586,411.245,171.386,34.870,156.543
C06939=1051.900,165.835,411.222,171.387,34.873,156.543
C06940=1051.905,166.084,411.199,171.389,34.875,156.544
C06941=1051.911,166.333,411.176,171.391,34.878,156.544
C06942=1051.917,166.581,411.153,171.393,34.880,156.545
C06943=1051.923,166.830,411.130,171.395,34.882,156.545
C06944=1051.929,167.080,411.109,171.398,34.885,156.545
C06945=1051.935,167.328,411.086,171.400,34.887,156.546
C06946=1051.940,167.577,411.063,171.402,34.890,156.546
C06947=1051.946,167.826,411.040,171.404,34.891,156.547
C06948=1051.952,168.075,411.017,171.406,34.894,156.547
C06949=1051.958,168.324,410.995,171.408,34.896,156.548
C06950=1051.964,168.573,410.972,171.411,34.899,156.548
C06951=1051.970,168.821,410.949,171.413,34.901,156.548
C06952=1051.975,169.070,410.926,171.415,34.903,156.549
C06953=1051.981,169.319,410.903,171.417,34.906,156.549
C06954=1051.988,169.568,410.881,171.419,34.908,156.550
C06955=1051.993,169.817,410.858,171.421,34.911,156.550
C06956=1051.999,170.066,410.835,171.423,34.913,156.551
C06957=1052.005,170.315,410.812,171.426,34.915,156.551
C06958=1052.011,170.563,410.789,171.428,34.918,156.551
C06959=1052.017,170.813,410.765,171.430,34.920,156.552
C06960=1052.024,171.061,410.742,171.432,34.923,156.552
C06961=1052.029,171.310,410.719,171.434,34.925,156.553
C06962=1052.035,171.559,410.697,171.436,34.927,156.553
C06963=1052.041,171.808,410.674,171.438,34.930,156.554
C06964=1052.047,172.057,410.651,171.441,34.932,156.554
C06965=1052.052,172.305,410.628,171.443,34.935,156.555
C06966=1052.059,172.554,410.605,171.445,34.937,156.555
C06967=1052.065,172.804,410.582,171.447,34.939,156.555
C06968=1052.071,173.053,410.559,171.449,34.942,156.556
C06969=1052.077,173.301,410.535,171.451,34.944,156.556
C06970=1052.083,173.550,410.512,171.453,34.947,156.557
C06971=1052.089,173.834,410.487,171.456,34.949,156.557
C06972=1052.097,174.119,410.459,171.458,34.952,156.558
C06973=1052.103,174.404,410.434,171.460,34.955,156.558
C06974=1052.110,174.688,410.407,171.463,34.957,156.559
C06975=1052.116,174.937,410.383,171.465,34.960,156.559
C06976=1052.123,175.186,410.361,171.467,34.962,156.560
C06977=1052.128,175.435,410.338,171.470,34.965,156.560
C06978=1052.134,175.684,410.315,171.472,34.967,156.560
C06979=1052.141,175.933,410.291,171.474,34.969,156.561
C06980=1052.146,176.182,410.268,171.476,34.972,156.561
C06981=1052.152,176.430,410.245,171.478,34.974,156.562
C06982=1052.158,176.679,410.222,171.480,34.977,156.562
C06983=1052.164,176.928,410.199,171.483,34.979,156.563
C06984=1052.170,177.177,410.175,171.485,34.981,156.563
C06985=1052.177,177.426,410.153,171.487,34.983,156.564
C06986=1052.183,177.674,410.129,171.489,34.986,156.564
C06987=1052.189,177.924,410.106,171.491,34.988,156.564
C06988=1052.195,178.173,410.083,171.493,34.991,156.565
C06989=1052.201,178.421,410.059,171.495,34.993,156.565
C06990=1052.207,178.670,410.036,171.498,34.995,156.566
C06991=1052.213,178.919,410.013,171.500,34.998,156.566
C06992=1052.219,179.168,409.990,171.503,35.000,156.567
C06993=1052.225,179.416,409.967,171.505,35.003,156.567
C06994=1052.231,179.665,409.943,171.507,35.005,156.568
C06995=1052.238,179.914,409.920,171.509,35.007,156.568
C06996=1052.244,180.162,409.897,171.511,35.010,156.568
C06997=1052.250,180.412,409.873,171.514,35.012,156.569
C06998=1052.256,180.661,409.850,171.516,35.015,156.569
C06999=1052.262,180.909,409.827,171.518,35.017,156.570
C07000=1052.268,181.159,409.803,171.520,35.020,156.570
C07001=1052.274,181.407,409.780,171.522,35.022,156.571
C07002=1052.280,181.656,409.757,171.524,35.024,156.571
C07003=1052.287,181.905,409.733,171.527,35.027,156.572
C07004=1052.292,182.154,409.710,171.530,35.029,156.572
C07005=1052.298,182.402,409.686,171.532,35.032,156.572
C07006=1052.305,182.652,409.663,171.534,35.034,156.573
C07007=1052.311,182.900,409.639,171.536,35.036,156.573
C07008=1052.317,183.149,409.616,171.538,35.038,156.574
C07009=1052.324,183.397,409.593,171.541,35.041,156.574
C07010=1052.330,183.646,409.569,171.543,35.043,156.575
C07011=1052.336,183.895,409.546,171.545,35.046,156.575
C07012=1052.342,184.144,409.522,171.547,35.048,156.576
C07013=1052.348,184.394,409.498,171.549,35.051,156.576
C07014=1052.354,184.642,409.474,171.552,35.053,156.576
C07015=1052.359,184.890,409.450,171.555,35.056,156.577
C07016=1052.366,185.139,409.426,171.557,35.058,156.577
C07017=1052.371,185.389,409.403,171.559,35.061,156.578
C07018=1052.377,185.637,409.379,171.561,35.063,156.578
C07019=1052.383,185.885,409.355,171.563,35.066,156.579
C07020=1052.389,186.134,409.331,171.565,35.069,156.579
C07021=1052.395,186.383,409.308,171.568,35.071,156.580
C07022=1052.400,186.632,409.284,171.570,35.074,156.580
C07023=1052.407,186.881,409.259,171.572,35.076,156.581
C07024=1052.412,187.129,409.235,171.574,35.079,156.581
C07025=1052.419,187.378,409.211,171.577,35.082,156.582
C07026=1052.423,187.628,409.188,171.579,35.084,156.582
C07027=1052.430,187.876,409.164,171.582,35.087,156.583
C07028=1052.435,188.125,409.139,171.584,35.089,156.583
C07029=1052.441,188.373,409.116,171.586,35.092,156.584
C07030=1052.447,188.622,409.091,171.588,35.094,156.584
C07031=1052.453,188.871,409.067,171.590,35.097,156.585
C07032=1052.459,189.119,409.044,171.593,35.100,156.585
C07033=1052.465,189.369,409.020,171.595,35.102,156.586
C07034=1052.471,189.618,408.996,171.598,35.105,156.586
C07035=1052.477,189.901,408.968,171.600,35.108,156.587
C07036=1052.484,190.186,408.941,171.602,35.111,156.587
C07037=1052.491,190.470,408.913,171.605,35.114,156.588
C07038=1052.498,190.755,408.885,171.608,35.117,156.588
C07039=1052.504,191.003,408.862,171.610,35.119,156.589
C07040=1052.510,191.252,408.837,171.613,35.122,156.589
C07041=1052.516,191.500,408.814,171.615,35.125,156.590
C07042=1052.521,191.749,408.789,171.617,35.127,156.590
C07043=1052.528,191.998,408.765,171.620,35.130,156.591
C07044=1052.533,192.247,408.741,171.622,35.132,156.591
C07045=1052.540,192.496,408.717,171.624,35.135,156.592
C07046=1052.545,192.744,408.693,171.627,35.138,156.592
C07047=1052.552,192.993,408.669,171.629,35.140,156.593
C07048=1052.557,193.242,408.644,171.632,35.143,156.593
C07049=1052.564,193.491,408.620,171.634,35.145,156.594
C07050=1052.569,193.739,408.596,171.636,35.148,156.594
C07051=1052.576,193.988,408.572,171.638,35.151,156.595
C07052=1052.581,194.237,408.548,171.641,35.153,156.595
C07053=1052.587,194.485,408.523,171.643,35.156,156.596
C07054=1052.594,194.734,408.499,171.646,35.158,156.596
C07055=1052.599,194.983,408.474,171.648,35.161,156.597
C07056=1052.606,195.232,408.450,171.650,35.164,156.597
C07057=1052.611,195.481,408.426,171.653,35.166,156.598
C07058=1052.618,195.730,408.402,171.655,35.169,156.598
C07059=1052.623,195.978,408.378,171.658,35.171,156.599
C07060=1052.630,196.227,408.353,171.660,35.174,156.599
C07061=1052.636,196.476,408.328,171.662,35.177,156.600
C07062=1052.642,196.724,408.305,171.665,35.179,156.600
C07063=1052.648,196.973,408.280,171.667,35.182,156.601
C07064=1052.653,197.221,408.255,171.669,35.184,156.601
C07065=1052.660,197.470,408.231,171.672,35.187,156.602
C07066=1052.666,197.720,408.206,171.674,35.190,156.602
C07067=1052.672,197.968,408.183,171.677,35.192,156.603
C07068=1052.678,198.217,408.157,171.679,35.195,156.603
C07069=1052.684,198.465,408.134,171.681,35.198,156.604
C07070=1052.690,198.714,408.109,171.684,35.200,156.604
C07071=1052.696,198.963,408.085,171.687,35.203,156.605
C07072=1052.702,199.211,408.060,171.689,35.206,156.605
C07073=1052.708,199.460,408.036,171.691,35.208,156.606
C07074=1052.715,199.709,408.011,171.693,35.211,156.606
C07075=1052.720,199.957,407.987,171.697,35.213,156.607
C07076=1052.727,200.206,407.962,171.699,35.216,156.607
C07077=1052.733,200.455,407.937,171.701,35.219,156.608
C07078=1052.739,200.704,407.913,171.703,35.221,156.608
C07079=1052.745,200.953,407.889,171.706,35.224,156.609
C07080=1052.751,201.201,407.864,171.709,35.227,156.609
C07081=1052.758,201.450,407.839,171.711,35.229,156.610
C07082=1052.764,201.698,407.815,171.713,35.232,156.610
C07083=1052.770,201.947,407.790,171.716,35.235,156.611
C07084=1052.776,202.196,407.765,171.718,35.237,156.611
C07085=1052.781,202.445,407.740,171.721,35.240,156.612
C07086=1052.787,202.693,407.715,171.723,35.243,156.612
C07087=1052.793,202.943,407.690,171.726,35.246,156.613
C07088=1052.800,203.190,407.666,171.728,35.248,156.613
C07089=1052.805,203.440,407.641,171.730,35.251,156.614
C07090=1052.812,203.688,407.616,171.733,35.254,156.614
C07091=1052.817,203.937,407.592,171.736,35.257,156.615
C07092=1052.823,204.186,407.566,171.738,35.259,156.615
C07093=1052.829,204.434,407.541,171.740,35.262,156.616
C07094=1052.835,204.683,407.516,171.742,35.265,156.616
C07095=1052.841,204.931,407.491,171.746,35.267,156.617
C07096=1052.847,205.181,407.467,171.748,35.271,156.618
C07097=1052.853,205.429,407.442,171.750,35.273,156.618
C07098=1052.859,205.678,407.416,171.753,35.276,156.619
C07099=1052.884,206.730,407.311,171.970,35.370,156.635
C07100=1052.892,206.974,407.286,171.971,35.373,156.636
C07101=1052.897,207.219,407.260,171.973,35.377,156.636
C07102=1052.904,207.465,407.235,171.976,35.380,156.637
C07103=1052.910,207.710,407.209,171.977,35.384,156.638
C07104=1052.916,207.955,407.184,171.979,35.388,156.639
C07105=1052.923,208.200,407.158,171.981,35.391,156.639
C07106=1052.929,208.445,407.133,171.983,35.394,156.640
C07107=1052.935,208.690,407.106,171.985,35.398,156.641
C07108=1052.941,208.939,407.081,171.986,35.402,156.641
C07109=1052.948,209.188,407.054,171.989,35.405,156.642
C07110=1052.954,209.436,407.028,171.991,35.409,156.643
C07111=1052.960,209.685,407.002,171.992,35.412,156.643
C07112=1052.966,209.933,406.976,171.995,35.416,156.644
C07113=1052.973,210.182,406.950,171.997,35.420,156.645
C07114=1052.979,210.431,406.924,171.998,35.423,156.646
C07115=1052.985,210.679,406.898,172.001,35.427,156.646
C07116=1052.993,210.927,406.871,172.003,35.430,156.647
C07117=1052.998,211.176,406.845,172.005,35.433,156.648
C07118=1053.005,211.424,406.819,172.006,35.437,156.648
C07119=1053.012,211.673,406.793,172.009,35.441,156.649
C07120=1053.017,211.922,406.766,172.011,35.444,156.650
C07121=1053.024,212.170,406.741,172.012,35.448,156.651
C07122=1053.030,212.419,406.714,172.015,35.452,156.651
C07123=1053.037,212.667,406.688,172.017,35.455,156.652
C07124=1053.042,212.916,406.661,172.018,35.459,156.653
C07125=1053.049,213.164,406.635,172.021,35.462,156.653
C07126=1053.055,213.413,406.608,172.023,35.466,156.654
C07127=1053.061,213.662,406.583,172.025,35.470,156.655
C07128=1053.068,213.911,406.556,172.027,35.473,156.656
C07129=1053.074,214.159,406.530,172.029,35.477,156.656
C07130=1053.080,214.407,406.503,172.031,35.480,156.657
C07131=1053.087,214.656,406.477,172.033,35.484,156.658
C07132=1053.093,214.904,406.450,172.035,35.487,156.658
C07133=1053.099,215.152,406.423,172.037,35.491,156.659
C07134=1053.106,215.401,406.397,172.039,35.494,156.660
C07135=1053.112,215.650,406.370,172.041,35.498,156.661
C07136=1053.118,215.898,406.345,172.043,35.501,156.661
C07137=1053.124,216.147,406.318,172.045,35.505,156.662
C07138=1053.131,216.395,406.292,172.048,35.509,156.663
C07139=1053.137,216.644,406.265,172.049,35.512,156.664
C07140=1053.144,216.892,406.239,172.051,35.516,156.664
C07141=1053.149,217.141,406.212,172.054,35.519,156.665
C07142=1053.156,217.390,406.185,172.056,35.523,156.666
C07143=1053.162,217.638,406.159,172.057,35.526,156.666
C07144=1053.169,217.887,406.132,172.060,35.530,156.667
C07145=1053.175,218.135,406.106,172.062,35.533,156.668
C07146=1053.181,218.384,406.079,172.064,35.537,156.668
C07147=1053.188,218.632,406.052,172.067,35.541,156.669
C07148=1053.194,218.880,406.026,172.068,35.544,156.670
C07149=1053.200,219.129,405.999,172.070,35.547,156.671
C07150=1053.207,219.377,405.972,172.073,35.551,156.671
C07151=1053.213,219.626,405.945,172.075,35.554,156.672
C07152=1053.220,219.874,405.919,172.076,35.558,156.673
C07153=1053.226,220.123,405.892,172.078,35.561,156.673
C07154=1053.232,220.372,405.866,172.081,35.565,156.674
C07155=1053.239,220.620,405.839,172.083,35.568,156.675
C07156=1053.245,220.868,405.812,172.085,35.572,156.676
C07157=1053.252,221.116,405.786,172.087,35.575,156.676
C07158=1053.258,221.364,405.759,172.089,35.579,156.677
C07159=1053.265,221.611,405.732,172.091,35.583,156.678
C07160=1053.270,221.860,405.705,172.094,35.586,156.678
C07161=1053.277,222.106,405.679,172.096,35.589,156.679
C07162=1053.283,222.354,405.651,172.097,35.593,156.680
C07163=1053.288,222.602,405.625,172.100,35.596,156.680
C07164=1053.296,222.851,405.598,172.102,35.600,156.681
C07165=1053.302,223.099,405.571,172.104,35.604,156.682
C07166=1053.308,223.348,405.544,172.107,35.607,156.683
C07167=1053.314,223.596,405.517,172.108,35.610,156.683
C07168=1053.320,223.845,405.490,172.110,35.614,156.684
C07169=1053.326,224.093,405.463,172.113,35.617,156.685
C07170=1053.333,224.342,405.436,172.115,35.621,156.685
C07171=1053.339,224.590,405.409,172.117,35.625,156.686
C07172=1053.346,224.839,405.382,172.120,35.628,156.687
C07173=1053.352,225.088,405.355,172.121,35.632,156.688
C07174=1053.358,225.335,405.328,172.123,35.635,156.688
C07175=1053.365,225.584,405.301,172.126,35.638,156.689
C07176=1053.371,225.832,405.273,172.128,35.642,156.690
C07177=1053.378,226.081,405.247,172.130,35.646,156.690
C07178=1053.384,226.329,405.220,172.133,35.649,156.691
C07179=1053.390,226.578,405.193,172.134,35.652,156.692
C07180=1053.397,226.827,405.165,172.136,35.656,156.693
C07181=1053.403,227.075,405.138,172.139,35.659,156.693
C07182=1053.409,227.324,405.111,172.141,35.663,156.694
C07183=1053.415,227.571,405.084,172.143,35.667,156.695
C07184=1053.422,227.820,405.057,172.145,35.670,156.695
C07185=1053.428,228.069,405.029,172.148,35.673,156.696
C07186=1053.435,228.317,405.003,172.150,35.677,156.697
C07187=1053.441,228.565,404.975,172.152,35.680,156.698
C07188=1053.448,228.814,404.948,172.154,35.683,156.698
C07189=1053.454,229.062,404.921,172.156,35.687,156.699
C07190=1053.460,229.311,404.894,172.158,35.690,156.700
C07191=1053.467,229.560,404.866,172.161,35.694,156.700
C07192=1053.473,229.807,404.839,172.163,35.698,156.701
C07193=1053.479,230.056,404.812,172.165,35.701,156.702
C07194=1053.486,230.304,404.784,172.168,35.704,156.702
C07195=1053.491,230.553,404.756,172.170,35.708,156.703
C07196=1053.498,230.802,404.729,172.172,35.711,156.704
C07197=1053.504,231.050,404.702,172.174,35.715,156.705
C07198=1053.511,231.298,404.674,172.176,35.719,156.705
C07199=1053.517,231.547,404.647,172.178,35.722,156.706
C07200=1053.523,231.795,404.620,172.181,35.725,156.707
C07201=1053.530,232.043,404.592,172.183,35.729,156.707
C07202=1053.536,232.292,404.565,172.186,35.732,156.708
C07203=1053.542,232.540,404.537,172.188,35.736,156.709
C07204=1053.548,232.789,404.509,172.190,35.739,156.709
C07205=1053.555,233.037,404.481,172.193,35.743,156.710
C07206=1053.561,233.286,404.455,172.195,35.746,156.711
C07207=1053.567,233.534,404.427,172.196,35.750,156.712
C07208=1053.574,233.783,404.399,172.199,35.753,156.712
C07209=1053.579,234.031,404.371,172.201,35.757,156.713
C07210=1053.586,234.279,404.344,172.203,35.760,156.714
C07211=1053.593,234.528,404.316,172.206,35.763,156.714
C07212=1053.598,234.772,404.289,172.208,35.767,156.715
C07213=1053.605,235.015,404.262,172.210,35.771,156.716
C07214=1053.611,235.260,404.235,172.213,35.774,156.717
C07215=1053.617,235.503,404.207,172.215,35.777,156.717
C07216=1053.623,235.747,404.180,172.217,35.781,156.718
C07217=1053.629,235.992,404.153,172.220,35.784,156.719
C07218=1053.635,236.235,404.125,172.222,35.787,156.719
C07219=1053.642,236.479,404.099,172.223,35.791,156.720
C07220=1053.648,236.728,404.070,172.226,35.795,156.721
C07221=1053.654,236.976,404.043,172.228,35.798,156.721
C07222=1053.661,237.225,404.015,172.230,35.801,156.722
C07223=1053.667,237.472,403.988,172.233,35.805,156.723
C07224=1053.673,237.721,403.959,172.235,35.808,156.724
C07225=1053.680,237.970,403.931,172.237,35.811,156.724
C07226=1053.686,238.218,403.904,172.240,35.815,156.725
C07227=1053.693,238.466,403.876,172.242,35.818,156.726
C07228=1053.699,238.715,403.848,172.244,35.822,156.726
C07229=1053.705,238.963,403.820,172.247,35.825,156.727
C07230=1053.712,239.211,403.793,172.249,35.829,156.728
C07231=1053.718,239.460,403.764,172.251,35.832,156.729
C07232=1053.725,239.709,403.737,172.254,35.836,156.729
C07233=1053.731,239.956,403.709,172.256,35.839,156.730
C07234=1053.737,240.205,403.681,172.258,35.842,156.731
C07235=1053.744,240.453,403.652,172.261,35.846,156.731
C07236=1053.749,240.702,403.624,172.263,35.849,156.732
C07237=1053.756,240.950,403.596,172.266,35.853,156.733
C07238=1053.763,241.199,403.569,172.268,35.856,156.733
C07239=1053.769,241.447,403.540,172.270,35.860,156.734
C07240=1053.775,241.696,403.513,172.273,35.863,156.735
C07241=1053.782,241.943,403.484,172.275,35.867,156.736
C07242=1053.788,242.192,403.456,172.277,35.870,156.736
C07243=1053.794,242.440,403.428,172.280,35.873,156.737
C07244=1053.800,242.689,403.400,172.282,35.877,156.738
C07245=1053.807,242.937,403.371,172.284,35.880,156.739
C07246=1053.813,243.185,403.343,172.287,35.884,156.739
C07247=1053.819,243.433,403.315,172.289,35.888,156.740
C07248=1053.825,243.682,403.286,172.291,35.891,156.741
C07249=1053.832,243.930,403.259,172.294,35.894,156.741
C07250=1053.838,244.179,403.230,172.297,35.898,156.742
C07251=1053.845,244.427,403.202,172.300,35.901,156.743
C07252=1053.850,244.675,403.174,172.302,35.905,156.744
C07253=1053.857,244.924,403.146,172.304,35.908,156.744
C07254=1053.863,245.172,403.117,172.307,35.911,156.745
C07255=1053.869,245.421,403.088,172.309,35.915,156.746
C07256=1053.876,245.669,403.061,172.311,35.919,156.746
C07257=1053.882,245.917,403.032,172.314,35.922,156.747
C07258=1053.888,246.165,403.004,172.316,35.925,156.748
C07259=1053.895,246.413,402.975,172.318,35.929,156.748
C07260=1053.901,246.662,402.947,172.321,35.932,156.749
C07261=1053.907,246.910,402.918,172.323,35.936,156.750
C07262=1053.913,247.159,402.890,172.326,35.939,156.751
C07263=1053.919,247.407,402.861,172.328,35.943,156.751
C07264=1053.925,247.656,402.832,172.330,35.946,156.752
C07265=1053.932,247.903,402.804,172.333,35.950,156.753
C07266=1053.938,248.152,402.775,172.335,35.954,156.754
C07267=1053.944,248.400,402.746,172.337,35.957,156.754
C07268=1053.950,248.641,402.718,172.340,35.960,156.755
C07269=1053.956,248.882,402.691,172.343,35.964,156.756
C07270=1053.961,249.122,402.663,172.345,35.967,156.757
C07271=1053.968,249.364,402.635,172.348,35.970,156.757
C07272=1053.974,249.605,402.607,172.350,35.974,156.758
C07273=1053.980,249.845,402.579,172.353,35.977,156.759
C07274=1053.986,250.087,402.552,172.355,35.980,156.759
C07275=1053.992,250.327,402.524,172.357,35.984,156.760
C07276=1053.999,250.575,402.495,172.360,35.987,156.761
C07277=1054.005,250.824,402.467,172.362,35.991,156.761
C07278=1054.011,251.072,402.437,172.364,35.994,156.762
C07279=1054.017,251.320,402.408,172.367,35.998,156.763
C07280=1054.023,251.569,402.380,172.369,36.001,156.764
C07281=1054.029,251.817,402.351,172.372,36.005,156.764
C07282=1054.036,252.065,402.322,172.374,36.008,156.765
C07283=1054.043,252.313,402.294,172.377,36.012,156.766
C07284=1054.049,252.561,402.265,172.380,36.015,156.766
C07285=1054.055,252.810,402.236,172.382,36.018,156.767
C07286=1054.061,253.058,402.207,172.384,36.022,156.768
C07287=1054.067,253.306,402.178,172.387,36.025,156.769
C07288=1054.074,253.554,402.149,172.389,36.029,156.769
